PROPERTY PUBLIC LeaderInfo : REFERENCE TO _GVSP_LEADER_PAYLOAD_IMAGE
GET
LeaderInfo REF= _LeaderInfo;
END_GET
END_PROPERTY

PROPERTY PUBLIC LocalIpAddress : REFERENCE TO _UDINT
GET
LocalIpAddress REF= _LocalIpAddress;
END_GET
END_PROPERTY

PROPERTY PUBLIC LocalUdpPort : REFERENCE TO _UINT
GET
LocalUdpPort REF= _LocalUdpPort;
END_GET
END_PROPERTY

METHOD PUBLIC MakeReferenceTo
VAR_INPUT
	ReferenceTarget : REFERENCE TO GVSP_IMAGE_INFO;
END_VAR
activeData REF= ReferenceTarget;
SetMemberReference();
END_METHOD

METHOD PROTECTED SetMemberReference
VAR_INPUT
END_VAR
_CameraIpAddress.MakeReferenceTo(activeData.CameraIpAddress);
_LocalIpAddress.MakeReferenceTo(activeData.LocalIpAddress);
_CameraUdpPort.MakeReferenceTo(activeData.CameraUdpPort);
_LocalUdpPort.MakeReferenceTo(activeData.LocalUdpPort);
_GvspChannelId.MakeReferenceTo(activeData.GvspChannelId);
_GevStatus.MakeReferenceTo(activeData.GevStatus);
_BlockId.MakeReferenceTo(activeData.BlockId);
_LeaderInfo.MakeReferenceTo(activeData.LeaderInfo);
END_METHOD

PROPERTY PUBLIC Size : UDINT
GET
Size := SIZEOF(activeData);
END_GET
END_PROPERTY

METHOD TryMakeReferenceTo : BOOL
VAR_INPUT
	Target : I_Datatype;
END_VAR
VAR
	targetAsStruct : I_StructuredDatatype;
	pTargetData : POINTER TO GVSP_IMAGE_INFO;
END_VAR
IF NOT Target.TryResolveAsStructuredDatatype(targetAsStruct) THEN
	RETURN;
END_IF

IF NOT (targetAsStruct.Identifier = Identifier) THEN
	RETURN;
END_IF

pTargetData := Target.Address;
activeData REF= pTargetData^;
SetMemberReference();
TryMakeReferenceTo := TRUE;
END_METHOD

PROPERTY PUBLIC Value : REFERENCE TO GVSP_IMAGE_INFO
GET
Value REF= activeData;
END_GET
END_PROPERTY

END_FUNCTION_BLOCK

// ---- Datatypes/Structs/_TcVnCodeGradesDM.TcPOU
{attribute 'linkalways'} 
{attribute 'no_explicit_call' := 'This FB is a CLASS and must be accessed using methods or properties'}
{attribute 'enable_dynamic_creation'}
FUNCTION_BLOCK _TcVnCodeGradesDM EXTENDS StructuredDatatypeBase
VAR
	localData : TcVnCodeGradesDM;
	activeData : REFERENCE TO TcVnCodeGradesDM REF= localData;
    _nDecode : _USINT(localdata.nDecode);
    _nSymbolContrast : _USINT(localdata.nSymbolContrast);
    _nModulation : _USINT(localdata.nModulation);
    _nReflectanceMargin : _USINT(localdata.nReflectanceMargin);
    _nFixedPatternDamage : _USINT(localdata.nFixedPatternDamage);
    _nAxialNonuniformity : _USINT(localdata.nAxialNonuniformity);
    _nGridNonuniformity : _USINT(localdata.nGridNonuniformity);
    _nUnusedErrorCorrection : _USINT(localdata.nUnusedErrorCorrection);
    _nOverall : _USINT(localdata.nOverall);
END_VAR

PROPERTY PUBLIC Address : PVOID
GET
Address := ADR(activeData);
END_GET
END_PROPERTY

METHOD PUBLIC ClearReference
VAR_INPUT
END_VAR
activeData REF= localData;
SetMemberReference();
END_METHOD

METHOD PUBLIC Clone : I_Datatype
VAR
    pClone : POINTER TO _TcVnCodeGradesDM;
END_VAR
pClone := __NEW(_TcVnCodeGradesDM());
pClone^.Value := Value;
Clone := pClone^;
END_METHOD

METHOD FB_init : BOOL
VAR_INPUT
	bInitRetains : BOOL; // if TRUE, the retain variables are initialized (warm start / cold start)
	bInCopyCode : BOOL;  // if TRUE, the instance afterwards gets moved into the copy code (online change)
END_VAR
SetMemberReference();
AddMember('nDecode', _nDecode);
AddMember('nSymbolContrast', _nSymbolContrast);
AddMember('nModulation', _nModulation);
AddMember('nReflectanceMargin', _nReflectanceMargin);
AddMember('nFixedPatternDamage', _nFixedPatternDamage);
AddMember('nAxialNonuniformity', _nAxialNonuniformity);
AddMember('nGridNonuniformity', _nGridNonuniformity);
AddMember('nUnusedErrorCorrection', _nUnusedErrorCorrection);
AddMember('nOverall', _nOverall);
END_METHOD

PROPERTY PUBLIC Identifier : T_MAXSTRING
GET
Identifier := 'TcVnCodeGradesDM';
END_GET
END_PROPERTY

METHOD PUBLIC MakeReferenceTo
VAR_INPUT
	ReferenceTarget : REFERENCE TO TcVnCodeGradesDM;
END_VAR
activeData REF= ReferenceTarget;
SetMemberReference();
END_METHOD

PROPERTY PUBLIC nAxialNonuniformity : REFERENCE TO _USINT
GET
nAxialNonuniformity REF= _nAxialNonuniformity;
END_GET
END_PROPERTY

PROPERTY PUBLIC nDecode : REFERENCE TO _USINT
GET
nDecode REF= _nDecode;
END_GET
END_PROPERTY

PROPERTY PUBLIC nFixedPatternDamage : REFERENCE TO _USINT
GET
nFixedPatternDamage REF= _nFixedPatternDamage;
END_GET
END_PROPERTY

PROPERTY PUBLIC nGridNonuniformity : REFERENCE TO _USINT
GET
nGridNonuniformity REF= _nGridNonuniformity;
END_GET
END_PROPERTY

PROPERTY PUBLIC nModulation : REFERENCE TO _USINT
GET
nModulation REF= _nModulation;
END_GET
END_PROPERTY

PROPERTY PUBLIC nOverall : REFERENCE TO _USINT
GET
nOverall REF= _nOverall;
END_GET
END_PROPERTY

PROPERTY PUBLIC nReflectanceMargin : REFERENCE TO _USINT
GET
nReflectanceMargin REF= _nReflectanceMargin;
END_GET
END_PROPERTY

PROPERTY PUBLIC nSymbolContrast : REFERENCE TO _USINT
GET
nSymbolContrast REF= _nSymbolContrast;
END_GET
END_PROPERTY

PROPERTY PUBLIC nUnusedErrorCorrection : REFERENCE TO _USINT
GET
nUnusedErrorCorrection REF= _nUnusedErrorCorrection;
END_GET
END_PROPERTY

METHOD PROTECTED SetMemberReference
VAR_INPUT
END_VAR
_nDecode.MakeReferenceTo(activeData.nDecode);
_nSymbolContrast.MakeReferenceTo(activeData.nSymbolContrast);
_nModulation.MakeReferenceTo(activeData.nModulation);
_nReflectanceMargin.MakeReferenceTo(activeData.nReflectanceMargin);
_nFixedPatternDamage.MakeReferenceTo(activeData.nFixedPatternDamage);
_nAxialNonuniformity.MakeReferenceTo(activeData.nAxialNonuniformity);
_nGridNonuniformity.MakeReferenceTo(activeData.nGridNonuniformity);
_nUnusedErrorCorrection.MakeReferenceTo(activeData.nUnusedErrorCorrection);
_nOverall.MakeReferenceTo(activeData.nOverall);
END_METHOD

PROPERTY PUBLIC Size : UDINT
GET
Size := SIZEOF(activeData);
END_GET
END_PROPERTY

METHOD TryMakeReferenceTo : BOOL
VAR_INPUT
	Target : I_Datatype;
END_VAR
VAR
	pTargetData : POINTER TO TcVnCodeGradesDM;
END_VAR
IF NOT IsEquivalentTo(Target) THEN
	RETURN;
END_IF

pTargetData := Target.Address;
activeData REF= pTargetData^;
SetMemberReference();
TryMakeReferenceTo := TRUE;
END_METHOD

PROPERTY PUBLIC Value : REFERENCE TO TcVnCodeGradesDM
GET
Value REF= activeData;
END_GET
END_PROPERTY

END_FUNCTION_BLOCK

// ---- Datatypes/Structs/_TcVnCodeGradesQR.TcPOU
{attribute 'linkalways'} 
{attribute 'no_explicit_call' := 'This FB is a CLASS and must be accessed using methods or properties'}
{attribute 'enable_dynamic_creation'}
FUNCTION_BLOCK _TcVnCodeGradesQR EXTENDS StructuredDatatypeBase
VAR
	localData : TcVnCodeGradesQR;
	activeData : REFERENCE TO TcVnCodeGradesQR REF= localData;
    _nDecode : _USINT(localdata.nDecode);
    _nSymbolContrast : _USINT(localdata.nSymbolContrast);
    _nModulation : _USINT(localdata.nModulation);
    _nReflectanceMargin : _USINT(localdata.nReflectanceMargin);
    _nFixedPatternDamage : _USINT(localdata.nFixedPatternDamage);
    _nAxialNonuniformity : _USINT(localdata.nAxialNonuniformity);
    _nGridNonuniformity : _USINT(localdata.nGridNonuniformity);
    _nUnusedErrorCorrection : _USINT(localdata.nUnusedErrorCorrection);
    _nFormatInfo : _USINT(localdata.nFormatInfo);
    _nVersionInfo : _USINT(localdata.nVersionInfo);
    _nOverall : _USINT(localdata.nOverall);
END_VAR

PROPERTY PUBLIC Address : PVOID
GET
Address := ADR(activeData);
END_GET
END_PROPERTY

METHOD PUBLIC ClearReference
VAR_INPUT
END_VAR
activeData REF= localData;
SetMemberReference();
END_METHOD

METHOD PUBLIC Clone : I_Datatype
VAR
    pClone : POINTER TO _TcVnCodeGradesQR;
END_VAR
pClone := __NEW(_TcVnCodeGradesQR());
pClone^.Value := Value;
Clone := pClone^;
END_METHOD

METHOD FB_init : BOOL
VAR_INPUT
	bInitRetains : BOOL; // if TRUE, the retain variables are initialized (warm start / cold start)
	bInCopyCode : BOOL;  // if TRUE, the instance afterwards gets moved into the copy code (online change)
END_VAR
SetMemberReference();
AddMember('nDecode', _nDecode);
AddMember('nSymbolContrast', _nSymbolContrast);
AddMember('nModulation', _nModulation);
AddMember('nReflectanceMargin', _nReflectanceMargin);
AddMember('nFixedPatternDamage', _nFixedPatternDamage);
AddMember('nAxialNonuniformity', _nAxialNonuniformity);
AddMember('nGridNonuniformity', _nGridNonuniformity);
AddMember('nUnusedErrorCorrection', _nUnusedErrorCorrection);
AddMember('nFormatInfo', _nFormatInfo);
AddMember('nVersionInfo', _nVersionInfo);
AddMember('nOverall', _nOverall);
END_METHOD

PROPERTY PUBLIC Identifier : T_MAXSTRING
GET
Identifier := 'TcVnCodeGradesQR';
END_GET
END_PROPERTY

METHOD PUBLIC MakeReferenceTo
VAR_INPUT
	ReferenceTarget : REFERENCE TO TcVnCodeGradesQR;
END_VAR
activeData REF= ReferenceTarget;
SetMemberReference();
END_METHOD

PROPERTY PUBLIC nAxialNonuniformity : REFERENCE TO _USINT
GET
nAxialNonuniformity REF= _nAxialNonuniformity;
END_GET
END_PROPERTY

PROPERTY PUBLIC nDecode : REFERENCE TO _USINT
GET
nDecode REF= _nDecode;
END_GET
END_PROPERTY

PROPERTY PUBLIC nFixedPatternDamage : REFERENCE TO _USINT
GET
nFixedPatternDamage REF= _nFixedPatternDamage;
END_GET
END_PROPERTY

PROPERTY PUBLIC nFormatInfo : REFERENCE TO _USINT
GET
nFormatInfo REF= _nFormatInfo;
END_GET
END_PROPERTY

PROPERTY PUBLIC nGridNonuniformity : REFERENCE TO _USINT
GET
nGridNonuniformity REF= _nGridNonuniformity;
END_GET
END_PROPERTY

PROPERTY PUBLIC nModulation : REFERENCE TO _USINT
GET
nModulation REF= _nModulation;
END_GET
END_PROPERTY

PROPERTY PUBLIC nOverall : REFERENCE TO _USINT
GET
nOverall REF= _nOverall;
END_GET
END_PROPERTY

PROPERTY PUBLIC nReflectanceMargin : REFERENCE TO _USINT
GET
nReflectanceMargin REF= _nReflectanceMargin;
END_GET
END_PROPERTY

PROPERTY PUBLIC nSymbolContrast : REFERENCE TO _USINT
GET
nSymbolContrast REF= _nSymbolContrast;
END_GET
END_PROPERTY

PROPERTY PUBLIC nUnusedErrorCorrection : REFERENCE TO _USINT
GET
nUnusedErrorCorrection REF= _nUnusedErrorCorrection;
END_GET
END_PROPERTY

PROPERTY PUBLIC nVersionInfo : REFERENCE TO _USINT
GET
nVersionInfo REF= _nVersionInfo;
END_GET
END_PROPERTY

METHOD PROTECTED SetMemberReference
VAR_INPUT
END_VAR
_nDecode.MakeReferenceTo(activeData.nDecode);
_nSymbolContrast.MakeReferenceTo(activeData.nSymbolContrast);
_nModulation.MakeReferenceTo(activeData.nModulation);
_nReflectanceMargin.MakeReferenceTo(activeData.nReflectanceMargin);
_nFixedPatternDamage.MakeReferenceTo(activeData.nFixedPatternDamage);
_nAxialNonuniformity.MakeReferenceTo(activeData.nAxialNonuniformity);
_nGridNonuniformity.MakeReferenceTo(activeData.nGridNonuniformity);
_nUnusedErrorCorrection.MakeReferenceTo(activeData.nUnusedErrorCorrection);
_nFormatInfo.MakeReferenceTo(activeData.nFormatInfo);
_nVersionInfo.MakeReferenceTo(activeData.nVersionInfo);
_nOverall.MakeReferenceTo(activeData.nOverall);
END_METHOD

PROPERTY PUBLIC Size : UDINT
GET
Size := SIZEOF(activeData);
END_GET
END_PROPERTY

METHOD TryMakeReferenceTo : BOOL
VAR_INPUT
	Target : I_Datatype;
END_VAR
VAR
	pTargetData : POINTER TO TcVnCodeGradesQR;
END_VAR
IF NOT IsEquivalentTo(Target) THEN
	RETURN;
END_IF

pTargetData := Target.Address;
activeData REF= pTargetData^;
SetMemberReference();
TryMakeReferenceTo := TRUE;
END_METHOD

PROPERTY PUBLIC Value : REFERENCE TO TcVnCodeGradesQR
GET
Value REF= activeData;
END_GET
END_PROPERTY

END_FUNCTION_BLOCK

// ---- Datatypes/Structs/_TcVnMoments.TcPOU
{attribute 'linkalways'} 
{attribute 'no_explicit_call' := 'This FB is a CLASS and must be accessed using methods or properties'}
{attribute 'enable_dynamic_creation'}
FUNCTION_BLOCK _TcVnMoments EXTENDS StructuredDatatypeBase
VAR
	localData : TcVnMoments;
	activeData : REFERENCE TO TcVnMoments REF= localData;
    _fM00 : _LREAL(localdata.fM00);
    _fM01 : _LREAL(localdata.fM01);
    _fM02 : _LREAL(localdata.fM02);
    _fM03 : _LREAL(localdata.fM03);
    _fM10 : _LREAL(localdata.fM10);
    _fM11 : _LREAL(localdata.fM11);
    _fM12 : _LREAL(localdata.fM12);
    _fM20 : _LREAL(localdata.fM20);
    _fM21 : _LREAL(localdata.fM21);
    _fM30 : _LREAL(localdata.fM30);
    _fMu02 : _LREAL(localdata.fMu02);
    _fMu03 : _LREAL(localdata.fMu03);
    _fMu11 : _LREAL(localdata.fMu11);
    _fMu12 : _LREAL(localdata.fMu12);
    _fMu20 : _LREAL(localdata.fMu20);
    _fMu21 : _LREAL(localdata.fMu21);
    _fMu30 : _LREAL(localdata.fMu30);
    _fNu02 : _LREAL(localdata.fNu02);
    _fNu03 : _LREAL(localdata.fNu03);
    _fNu11 : _LREAL(localdata.fNu11);
    _fNu12 : _LREAL(localdata.fNu12);
    _fNu20 : _LREAL(localdata.fNu20);
    _fNu21 : _LREAL(localdata.fNu21);
    _fNu30 : _LREAL(localdata.fNu30);
END_VAR

PROPERTY PUBLIC Address : PVOID
GET
Address := ADR(activeData);
END_GET
END_PROPERTY

METHOD PUBLIC ClearReference
VAR_INPUT
END_VAR
activeData REF= localData;
SetMemberReference();
END_METHOD

METHOD PUBLIC Clone : I_Datatype
VAR
    pClone : POINTER TO _TcVnMoments;
END_VAR
pClone := __NEW(_TcVnMoments());
pClone^.Value := Value;
Clone := pClone^;
END_METHOD

METHOD FB_init : BOOL
VAR_INPUT
	bInitRetains : BOOL; // if TRUE, the retain variables are initialized (warm start / cold start)
	bInCopyCode : BOOL;  // if TRUE, the instance afterwards gets moved into the copy code (online change)
END_VAR
SetMemberReference();
AddMember('fM00', _fM00);
AddMember('fM01', _fM01);
AddMember('fM02', _fM02);
AddMember('fM03', _fM03);
AddMember('fM10', _fM10);
AddMember('fM11', _fM11);
AddMember('fM12', _fM12);
AddMember('fM20', _fM20);
AddMember('fM21', _fM21);
AddMember('fM30', _fM30);
AddMember('fMu02', _fMu02);
AddMember('fMu03', _fMu03);
AddMember('fMu11', _fMu11);
AddMember('fMu12', _fMu12);
AddMember('fMu20', _fMu20);
AddMember('fMu21', _fMu21);
AddMember('fMu30', _fMu30);
AddMember('fNu02', _fNu02);
AddMember('fNu03', _fNu03);
AddMember('fNu11', _fNu11);
AddMember('fNu12', _fNu12);
AddMember('fNu20', _fNu20);
AddMember('fNu21', _fNu21);
AddMember('fNu30', _fNu30);
END_METHOD

PROPERTY PUBLIC fM00 : REFERENCE TO _LREAL
GET
fM00 REF= _fM00;
END_GET
END_PROPERTY

PROPERTY PUBLIC fM01 : REFERENCE TO _LREAL
GET
fM01 REF= _fM01;
END_GET
END_PROPERTY

PROPERTY PUBLIC fM02 : REFERENCE TO _LREAL
GET
fM02 REF= _fM02;
END_GET
END_PROPERTY

PROPERTY PUBLIC fM03 : REFERENCE TO _LREAL
GET
fM03 REF= _fM03;
END_GET
END_PROPERTY

PROPERTY PUBLIC fM10 : REFERENCE TO _LREAL
GET
fM10 REF= _fM10;
END_GET
END_PROPERTY

PROPERTY PUBLIC fM11 : REFERENCE TO _LREAL
GET
fM11 REF= _fM11;
END_GET
END_PROPERTY

PROPERTY PUBLIC fM12 : REFERENCE TO _LREAL
GET
fM12 REF= _fM12;
END_GET
END_PROPERTY

PROPERTY PUBLIC fM20 : REFERENCE TO _LREAL
GET
fM20 REF= _fM20;
END_GET
END_PROPERTY

PROPERTY PUBLIC fM21 : REFERENCE TO _LREAL
GET
fM21 REF= _fM21;
END_GET
END_PROPERTY

PROPERTY PUBLIC fM30 : REFERENCE TO _LREAL
GET
fM30 REF= _fM30;
END_GET
END_PROPERTY

PROPERTY PUBLIC fMu02 : REFERENCE TO _LREAL
GET
fMu02 REF= _fMu02;
END_GET
END_PROPERTY

PROPERTY PUBLIC fMu03 : REFERENCE TO _LREAL
GET
fMu03 REF= _fMu03;
END_GET
END_PROPERTY

PROPERTY PUBLIC fMu11 : REFERENCE TO _LREAL
GET
fMu11 REF= _fMu11;
END_GET
END_PROPERTY

PROPERTY PUBLIC fMu12 : REFERENCE TO _LREAL
GET
fMu12 REF= _fMu12;
END_GET
END_PROPERTY

PROPERTY PUBLIC fMu20 : REFERENCE TO _LREAL
GET
fMu20 REF= _fMu20;
END_GET
END_PROPERTY

PROPERTY PUBLIC fMu21 : REFERENCE TO _LREAL
GET
fMu21 REF= _fMu21;
END_GET
END_PROPERTY

PROPERTY PUBLIC fMu30 : REFERENCE TO _LREAL
GET
fMu30 REF= _fMu30;
END_GET
END_PROPERTY

PROPERTY PUBLIC fNu02 : REFERENCE TO _LREAL
GET
fNu02 REF= _fNu02;
END_GET
END_PROPERTY

PROPERTY PUBLIC fNu03 : REFERENCE TO _LREAL
GET
fNu03 REF= _fNu03;
END_GET
END_PROPERTY

PROPERTY PUBLIC fNu11 : REFERENCE TO _LREAL
GET
fNu11 REF= _fNu11;
END_GET
END_PROPERTY

PROPERTY PUBLIC fNu12 : REFERENCE TO _LREAL
GET
fNu12 REF= _fNu12;
END_GET
END_PROPERTY

PROPERTY PUBLIC fNu20 : REFERENCE TO _LREAL
GET
fNu20 REF= _fNu20;
END_GET
END_PROPERTY

PROPERTY PUBLIC fNu21 : REFERENCE TO _LREAL
GET
fNu21 REF= _fNu21;
END_GET
END_PROPERTY

PROPERTY PUBLIC fNu30 : REFERENCE TO _LREAL
GET
fNu30 REF= _fNu30;
END_GET
END_PROPERTY

PROPERTY PUBLIC Identifier : T_MAXSTRING
GET
Identifier := 'TcVnMoments';
END_GET
END_PROPERTY

METHOD PUBLIC MakeReferenceTo
VAR_INPUT
	ReferenceTarget : REFERENCE TO TcVnMoments;
END_VAR
activeData REF= ReferenceTarget;
SetMemberReference();
END_METHOD

METHOD PROTECTED SetMemberReference
VAR_INPUT
END_VAR
_fM00.MakeReferenceTo(activeData.fM00);
_fM01.MakeReferenceTo(activeData.fM01);
_fM02.MakeReferenceTo(activeData.fM02);
_fM03.MakeReferenceTo(activeData.fM03);
_fM10.MakeReferenceTo(activeData.fM10);
_fM11.MakeReferenceTo(activeData.fM11);
_fM12.MakeReferenceTo(activeData.fM12);
_fM20.MakeReferenceTo(activeData.fM20);
_fM21.MakeReferenceTo(activeData.fM21);
_fM30.MakeReferenceTo(activeData.fM30);
_fMu02.MakeReferenceTo(activeData.fMu02);
_fMu03.MakeReferenceTo(activeData.fMu03);
_fMu11.MakeReferenceTo(activeData.fMu11);
_fMu12.MakeReferenceTo(activeData.fMu12);
_fMu20.MakeReferenceTo(activeData.fMu20);
_fMu21.MakeReferenceTo(activeData.fMu21);
_fMu30.MakeReferenceTo(activeData.fMu30);
_fNu02.MakeReferenceTo(activeData.fNu02);
_fNu03.MakeReferenceTo(activeData.fNu03);
_fNu11.MakeReferenceTo(activeData.fNu11);
_fNu12.MakeReferenceTo(activeData.fNu12);
_fNu20.MakeReferenceTo(activeData.fNu20);
_fNu21.MakeReferenceTo(activeData.fNu21);
_fNu30.MakeReferenceTo(activeData.fNu30);
END_METHOD

PROPERTY PUBLIC Size : UDINT
GET
Size := SIZEOF(activeData);
END_GET
END_PROPERTY

METHOD TryMakeReferenceTo : BOOL
VAR_INPUT
	Target : I_Datatype;
END_VAR
VAR
	pTargetData : POINTER TO TcVnMoments;
END_VAR
IF NOT IsEquivalentTo(Target) THEN
	RETURN;
END_IF

pTargetData := Target.Address;
activeData REF= pTargetData^;
SetMemberReference();
TryMakeReferenceTo := TRUE;
END_METHOD

PROPERTY PUBLIC Value : REFERENCE TO TcVnMoments
GET
Value REF= activeData;
END_GET
END_PROPERTY

END_FUNCTION_BLOCK

// ---- Datatypes/Structs/_TcVnDMatch.TcPOU
{attribute 'linkalways'} 
{attribute 'no_explicit_call' := 'This FB is a CLASS and must be accessed using methods or properties'}
{attribute 'enable_dynamic_creation'}
FUNCTION_BLOCK _TcVnDMatch EXTENDS StructuredDatatypeBase
VAR
	localData : TcVnDMatch;
	activeData : REFERENCE TO TcVnDMatch REF= localData;
    _nQueryIdx : _DINT(localdata.nQueryIdx);
    _nTrainIdx : _DINT(localdata.nTrainIdx);
    _nImageIdx : _DINT(localdata.nImageIdx);
    _fDistance : _REAL(localdata.fDistance);
END_VAR

PROPERTY PUBLIC Address : PVOID
GET
Address := ADR(activeData);
END_GET
END_PROPERTY

METHOD PUBLIC ClearReference
VAR_INPUT
END_VAR
activeData REF= localData;
SetMemberReference();
END_METHOD

METHOD PUBLIC Clone : I_Datatype
VAR
    pClone : POINTER TO _TcVnDMatch;
END_VAR
pClone := __NEW(_TcVnDMatch());
pClone^.Value := Value;
Clone := pClone^;
END_METHOD

METHOD FB_init : BOOL
VAR_INPUT
	bInitRetains : BOOL; // if TRUE, the retain variables are initialized (warm start / cold start)
	bInCopyCode : BOOL;  // if TRUE, the instance afterwards gets moved into the copy code (online change)
END_VAR
SetMemberReference();
AddMember('nQueryIdx', _nQueryIdx);
AddMember('nTrainIdx', _nTrainIdx);
AddMember('nImageIdx', _nImageIdx);
AddMember('fDistance', _fDistance);
END_METHOD

PROPERTY PUBLIC fDistance : REFERENCE TO _REAL
GET
fDistance REF= _fDistance;
END_GET
END_PROPERTY

PROPERTY PUBLIC Identifier : T_MAXSTRING
GET
Identifier := 'TcVnDMatch';
END_GET
END_PROPERTY

METHOD PUBLIC MakeReferenceTo
VAR_INPUT
	ReferenceTarget : REFERENCE TO TcVnDMatch;
END_VAR
activeData REF= ReferenceTarget;
SetMemberReference();
END_METHOD

PROPERTY PUBLIC nImageIdx : REFERENCE TO _DINT
GET
nImageIdx REF= _nImageIdx;
END_GET
END_PROPERTY

PROPERTY PUBLIC nQueryIdx : REFERENCE TO _DINT
GET
nQueryIdx REF= _nQueryIdx;
END_GET
END_PROPERTY

PROPERTY PUBLIC nTrainIdx : REFERENCE TO _DINT
GET
nTrainIdx REF= _nTrainIdx;
END_GET
END_PROPERTY

METHOD PROTECTED SetMemberReference
VAR_INPUT
END_VAR
_nQueryIdx.MakeReferenceTo(activeData.nQueryIdx);
_nTrainIdx.MakeReferenceTo(activeData.nTrainIdx);
_nImageIdx.MakeReferenceTo(activeData.nImageIdx);
_fDistance.MakeReferenceTo(activeData.fDistance);
END_METHOD

PROPERTY PUBLIC Size : UDINT
GET
Size := SIZEOF(activeData);
END_GET
END_PROPERTY

METHOD TryMakeReferenceTo : BOOL
VAR_INPUT
	Target : I_Datatype;
END_VAR
VAR
	targetAsStruct : I_StructuredDatatype;
	pTargetData : POINTER TO TcVnDMatch;
END_VAR
IF NOT Target.TryResolveAsStructuredDatatype(targetAsStruct) THEN
	RETURN;
END_IF

IF NOT (targetAsStruct.Identifier = Identifier) THEN
	RETURN;
END_IF

pTargetData := Target.Address;
activeData REF= pTargetData^;
SetMemberReference();
TryMakeReferenceTo := TRUE;
END_METHOD

PROPERTY PUBLIC Value : REFERENCE TO TcVnDMatch
GET
Value REF= activeData;
END_GET
END_PROPERTY

END_FUNCTION_BLOCK

// ---- Datatypes/Structs/_TcVnCodeGrades1D.TcPOU
{attribute 'linkalways'} 
{attribute 'no_explicit_call' := 'This FB is a CLASS and must be accessed using methods or properties'}
{attribute 'enable_dynamic_creation'}
FUNCTION_BLOCK _TcVnCodeGrades1D EXTENDS StructuredDatatypeBase
VAR
	localData : TcVnCodeGrades1D;
	activeData : REFERENCE TO TcVnCodeGrades1D REF= localData;
    _fDecode : _REAL(localdata.fDecode);
    _fSymbolContrast : _REAL(localdata.fSymbolContrast);
    _fMinReflectance : _REAL(localdata.fMinReflectance);
    _fMinEdgeContrast : _REAL(localdata.fMinEdgeContrast);
    _fModulation : _REAL(localdata.fModulation);
    _fDefects : _REAL(localdata.fDefects);
    _fDecodability : _REAL(localdata.fDecodability);
    _fOverall : _REAL(localdata.fOverall);
END_VAR

PROPERTY PUBLIC Address : PVOID
GET
Address := ADR(activeData);
END_GET
END_PROPERTY

METHOD PUBLIC ClearReference
VAR_INPUT
END_VAR
activeData REF= localData;
SetMemberReference();
END_METHOD

METHOD PUBLIC Clone : I_Datatype
VAR
    pClone : POINTER TO _TcVnCodeGrades1D;
END_VAR
pClone := __NEW(_TcVnCodeGrades1D());
pClone^.Value := Value;
Clone := pClone^;
END_METHOD

METHOD FB_init : BOOL
VAR_INPUT
	bInitRetains : BOOL; // if TRUE, the retain variables are initialized (warm start / cold start)
	bInCopyCode : BOOL;  // if TRUE, the instance afterwards gets moved into the copy code (online change)
END_VAR
SetMemberReference();
AddMember('fDecode', _fDecode);
AddMember('fSymbolContrast', _fSymbolContrast);
AddMember('fMinReflectance', _fMinReflectance);
AddMember('fMinEdgeContrast', _fMinEdgeContrast);
AddMember('fModulation', _fModulation);
AddMember('fDefects', _fDefects);
AddMember('fDecodability', _fDecodability);
AddMember('fOverall', _fOverall);
END_METHOD

PROPERTY PUBLIC fDecodability : REFERENCE TO _REAL
GET
fDecodability REF= _fDecodability;
END_GET
END_PROPERTY

PROPERTY PUBLIC fDecode : REFERENCE TO _REAL
GET
fDecode REF= _fDecode;
END_GET
END_PROPERTY

PROPERTY PUBLIC fDefects : REFERENCE TO _REAL
GET
fDefects REF= _fDefects;
END_GET
END_PROPERTY

PROPERTY PUBLIC fMinEdgeContrast : REFERENCE TO _REAL
GET
fMinEdgeContrast REF= _fMinEdgeContrast;
END_GET
END_PROPERTY

PROPERTY PUBLIC fMinReflectance : REFERENCE TO _REAL
GET
fMinReflectance REF= _fMinReflectance;
END_GET
END_PROPERTY

PROPERTY PUBLIC fModulation : REFERENCE TO _REAL
GET
fModulation REF= _fModulation;
END_GET
END_PROPERTY

PROPERTY PUBLIC fOverall : REFERENCE TO _REAL
GET
fOverall REF= _fOverall;
END_GET
END_PROPERTY

PROPERTY PUBLIC fSymbolContrast : REFERENCE TO _REAL
GET
fSymbolContrast REF= _fSymbolContrast;
END_GET
END_PROPERTY

PROPERTY PUBLIC Identifier : T_MAXSTRING
GET
Identifier := 'TcVnCodeGrades1D';
END_GET
END_PROPERTY

METHOD PUBLIC MakeReferenceTo
VAR_INPUT
	ReferenceTarget : REFERENCE TO TcVnCodeGrades1D;
END_VAR
activeData REF= ReferenceTarget;
SetMemberReference();
END_METHOD

METHOD PROTECTED SetMemberReference
VAR_INPUT
END_VAR
_fDecode.MakeReferenceTo(activeData.fDecode);
_fSymbolContrast.MakeReferenceTo(activeData.fSymbolContrast);
_fMinReflectance.MakeReferenceTo(activeData.fMinReflectance);
_fMinEdgeContrast.MakeReferenceTo(activeData.fMinEdgeContrast);
_fModulation.MakeReferenceTo(activeData.fModulation);
_fDefects.MakeReferenceTo(activeData.fDefects);
_fDecodability.MakeReferenceTo(activeData.fDecodability);
_fOverall.MakeReferenceTo(activeData.fOverall);
END_METHOD

PROPERTY PUBLIC Size : UDINT
GET
Size := SIZEOF(activeData);
END_GET
END_PROPERTY

METHOD TryMakeReferenceTo : BOOL
VAR_INPUT
	Target : I_Datatype;
END_VAR
VAR
	pTargetData : POINTER TO TcVnCodeGrades1D;
END_VAR
IF NOT IsEquivalentTo(Target) THEN
	RETURN;
END_IF

pTargetData := Target.Address;
activeData REF= pTargetData^;
SetMemberReference();
TryMakeReferenceTo := TRUE;
END_METHOD

PROPERTY PUBLIC Value : REFERENCE TO TcVnCodeGrades1D
GET
Value REF= activeData;
END_GET
END_PROPERTY

END_FUNCTION_BLOCK

// ---- Datatypes/Structs/_TcVnMatrix.TcPOU
{attribute 'linkalways'} 
{attribute 'no_explicit_call' := 'This FB is a CLASS and must be accessed using methods or properties'}
{attribute 'enable_dynamic_creation'}
FUNCTION_BLOCK _TcVnMatrix EXTENDS StructuredDatatypeBase
VAR
	localData : TcVnMatrix;
	activeData : REFERENCE TO TcVnMatrix REF= localData;
	_nRows : _UDINT(localData.nRows);
    _nCols : _UDINT(localData.nCols);
    _eType : _ETcVnElementType(localData.eType);
    _pData : _PVOID(localData.pData);
END_VAR

PROPERTY PUBLIC Address : PVOID
GET
Address := ADR(activeData);
END_GET
END_PROPERTY

METHOD PUBLIC ClearReference
VAR_INPUT
END_VAR
activeData REF= localData;
SetMemberReference();
END_METHOD

METHOD PUBLIC Clone : I_Datatype
VAR
    pClone : POINTER TO _TcVnMatrix;
END_VAR
pClone := __NEW(_TcVnMatrix());
pClone^.Value := Value;
Clone := pClone^;
END_METHOD

PROPERTY PUBLIC eType : REFERENCE TO _ETcVnElementType
GET
eType REF= _eType;
END_GET
END_PROPERTY

METHOD FB_init : BOOL
VAR_INPUT
	bInitRetains : BOOL; // if TRUE, the retain variables are initialized (warm start / cold start)
	bInCopyCode : BOOL;  // if TRUE, the instance afterwards gets moved into the copy code (online change)
END_VAR
SetMemberReference();
AddMember('nRows', _nRows);
AddMember('nCols', _nCols);
AddMember('eType', _eType);
AddMember('pData', _pData);
END_METHOD

PROPERTY PUBLIC Identifier : T_MAXSTRING
GET
Identifier := 'TcVnMatrix';
END_GET
END_PROPERTY

METHOD PUBLIC MakeReferenceTo
VAR_INPUT
	ReferenceTarget : REFERENCE TO TcVnMatrix;
END_VAR
activeData REF= ReferenceTarget;
SetMemberReference();
END_METHOD

PROPERTY PUBLIC nCols : REFERENCE TO _UDINT
GET
nCols REF= _nCols;
END_GET
END_PROPERTY

PROPERTY PUBLIC nRows : REFERENCE TO _UDINT
GET
nRows REF= _nRows;
END_GET
END_PROPERTY

PROPERTY PUBLIC pData : REFERENCE TO _PVOID
GET
pData REF= _pData;
END_GET
END_PROPERTY

METHOD PROTECTED SetMemberReference
VAR_INPUT
END_VAR
_nRows.MakeReferenceTo(activeData.nRows);
_nCols.MakeReferenceTo(activeData.nCols);
_eType.MakeReferenceTo(activeData.eType);
_pData.MakeReferenceTo(activeData.pData);
END_METHOD

PROPERTY PUBLIC Size : UDINT
GET
Size := SIZEOF(activeData);
END_GET
END_PROPERTY

METHOD TryMakeReferenceTo : BOOL
VAR_INPUT
	Target : I_Datatype;
END_VAR
VAR
	pTargetData : POINTER TO TcVnMatrix;
END_VAR
IF NOT IsEquivalentTo(Target) THEN
	RETURN;
END_IF

pTargetData := Target.Address;
activeData REF= pTargetData^;
SetMemberReference();
TryMakeReferenceTo := TRUE;
END_METHOD

PROPERTY PUBLIC Value : REFERENCE TO TcVnMatrix
GET
Value REF= activeData;
END_GET
END_PROPERTY

END_FUNCTION_BLOCK

// ---- Datatypes/Structs/_TcVnParamsMSER.TcPOU
{attribute 'linkalways'} 
{attribute 'no_explicit_call' := 'This FB is a CLASS and must be accessed using methods or properties'}
{attribute 'enable_dynamic_creation'}
FUNCTION_BLOCK _TcVnParamsMSER EXTENDS StructuredDatatypeBase
VAR
	localData : TcVnParamsMSER;
	activeData : REFERENCE TO TcVnParamsMSER REF= localData;
	_nDelta : _DINT(localData.nDelta);
    _nMinArea : _UDINT(localData.nMinArea);
	_nMaxArea : _UDINT(localData.nMaxArea);
	_fMaxVariation : _LREAL(localData.fMaxVariation);
	_fMinDiversity : _LREAL(localData.fMinDiversity);
	_nMaxEvolution : _UDINT(localData.nMaxEvolution);
    _fAreaThreshold : _LREAL(localData.fAreaThreshold);
    _fMinMargin : _LREAL(localData.fMinMargin);
    _nEdgeBlurSize : _UDINT(localData.nEdgeBlurSize);
END_VAR

PROPERTY PUBLIC Address : PVOID
GET
Address := ADR(activeData);
END_GET
END_PROPERTY

METHOD PUBLIC ClearReference
VAR_INPUT
END_VAR
activeData REF= localData;
SetMemberReference();
END_METHOD

METHOD PUBLIC Clone : I_Datatype
VAR
    pClone : POINTER TO _TcVnParamsMSER;
END_VAR
pClone := __NEW(_TcVnParamsMSER());
pClone^.Value := Value;
Clone := pClone^;
END_METHOD

PROPERTY PUBLIC fAreaThreshold : REFERENCE TO _LREAL
GET
fAreaThreshold REF= _fAreaThreshold;
END_GET
END_PROPERTY

METHOD FB_init : BOOL
VAR_INPUT
	bInitRetains : BOOL; // if TRUE, the retain variables are initialized (warm start / cold start)
	bInCopyCode : BOOL;  // if TRUE, the instance afterwards gets moved into the copy code (online change)
END_VAR
SetMemberReference();
AddMember('nDelta', _nDelta);
AddMember('nMinArea', _nMinArea);
AddMember('nMaxArea', _nMaxArea);
AddMember('fMaxVariation', _fMaxVariation);
AddMember('fMinDiversity', _fMinDiversity);
AddMember('nMaxEvolution', _nMaxEvolution);
AddMember('fAreaThreshold', _fAreaThreshold);
AddMember('fMinMargin', _fMinMargin);
AddMember('nEdgeBlurSize', _nEdgeBlurSize);
END_METHOD

PROPERTY PUBLIC fMaxVariation : REFERENCE TO _LREAL
GET
fMaxVariation REF= _fMaxVariation;
END_GET
END_PROPERTY

PROPERTY PUBLIC fMinDiversity : REFERENCE TO _LREAL
GET
fMinDiversity REF= _fMinDiversity;
END_GET
END_PROPERTY

PROPERTY PUBLIC fMinMargin : REFERENCE TO _LREAL
GET
fMinMargin REF= _fMinMargin;
END_GET
END_PROPERTY

PROPERTY PUBLIC Identifier : T_MAXSTRING
GET
Identifier := 'TcVnParamsMSER';
END_GET
END_PROPERTY

METHOD PUBLIC MakeReferenceTo
VAR_INPUT
	ReferenceTarget : REFERENCE TO TcVnParamsMSER;
END_VAR
activeData REF= ReferenceTarget;
SetMemberReference();
END_METHOD

PROPERTY PUBLIC nDelta : REFERENCE TO _DINT
GET
nDelta REF= _nDelta;
END_GET
END_PROPERTY

PROPERTY PUBLIC nEdgeBlurSize : REFERENCE TO _UDINT
GET
nEdgeBlurSize REF= _nEdgeBlurSize;
END_GET
END_PROPERTY

PROPERTY PUBLIC nMaxArea : REFERENCE TO _UDINT
GET
nMaxArea REF= _nMaxArea;
END_GET
END_PROPERTY

PROPERTY PUBLIC nMaxEvolution : REFERENCE TO _UDINT
GET
nMaxEvolution REF= _nMaxEvolution;
END_GET
END_PROPERTY

PROPERTY PUBLIC nMinArea : REFERENCE TO _UDINT
GET
nMinArea REF= _nMinArea;
END_GET
END_PROPERTY

METHOD PROTECTED SetMemberReference
VAR_INPUT
END_VAR
_nDelta.MakeReferenceTo(activeData.nDelta);
_nMinArea.MakeReferenceTo(activeData.nMinArea);
_nMaxArea.MakeReferenceTo(activeData.nMaxArea);
_fMaxVariation.MakeReferenceTo(activeData.fMaxVariation);
_fMinDiversity.MakeReferenceTo(activeData.fMinDiversity);
_nMaxEvolution.MakeReferenceTo(activeData.nMaxEvolution);
_fAreaThreshold.MakeReferenceTo(activeData.fAreaThreshold);
_fMinMargin.MakeReferenceTo(activeData.fMinMargin);
_nEdgeBlurSize.MakeReferenceTo(activeData.nEdgeBlurSize);
END_METHOD

PROPERTY PUBLIC Size : UDINT
GET
Size := SIZEOF(activeData);
END_GET
END_PROPERTY

METHOD TryMakeReferenceTo : BOOL
VAR_INPUT
	Target : I_Datatype;
END_VAR
VAR
	pTargetData : POINTER TO TcVnParamsMSER;
END_VAR
IF NOT IsEquivalentTo(Target) THEN
	RETURN;
END_IF

pTargetData := Target.Address;
activeData REF= pTargetData^;
SetMemberReference();
TryMakeReferenceTo := TRUE;
END_METHOD

PROPERTY PUBLIC Value : REFERENCE TO TcVnParamsMSER
GET
Value REF= activeData;
END_GET
END_PROPERTY

END_FUNCTION_BLOCK

// ---- Datatypes/Structs/_TcVnParamsAKAZE.TcPOU
{attribute 'linkalways'} 
{attribute 'no_explicit_call' := 'This FB is a CLASS and must be accessed using methods or properties'}
{attribute 'enable_dynamic_creation'}
FUNCTION_BLOCK _TcVnParamsAKAZE EXTENDS StructuredDatatypeBase
VAR
	localData : TcVnParamsAKAZE;
	activeData : REFERENCE TO TcVnParamsAKAZE REF= localData;
    _eDescrType     : _ETcVnFeatureDescriptorTypeAKAZE(localdata.eDescrType);
    _nDescrSize     : _UDINT(localdata.nDescrSize);
    _nDescrChannels : _UDINT(localdata.nDescrChannels);
    _fThreshold     : _REAL(localdata.fThreshold);
    _nOctaves       : _UDINT(localdata.nOctaves);
    _nOctaveLayers  : _UDINT(localdata.nOctaveLayers);
    _eDiffusivity   : _ETcVnDiffusivityTypeKAZE(localdata.eDiffusivity);
END_VAR

PROPERTY PUBLIC Address : PVOID
GET
Address := ADR(activeData);
END_GET
END_PROPERTY

METHOD PUBLIC ClearReference
VAR_INPUT
END_VAR
activeData REF= localData;
SetMemberReference();
END_METHOD

METHOD PUBLIC Clone : I_Datatype
VAR
    pClone : POINTER TO _TcVnParamsAKAZE;
END_VAR
pClone := __NEW(_TcVnParamsAKAZE());
pClone^.Value := Value;
Clone := pClone^;
END_METHOD

PROPERTY PUBLIC eDescrType : REFERENCE TO _ETcVnFeatureDescriptorTypeAKAZE
GET
eDescrType REF= _eDescrType;
END_GET
END_PROPERTY

PROPERTY PUBLIC eDiffusivity : REFERENCE TO _ETcVnDiffusivityTypeKAZE
GET
eDiffusivity REF= _eDiffusivity;
END_GET
END_PROPERTY

METHOD FB_init : BOOL
VAR_INPUT
	bInitRetains : BOOL; // if TRUE, the retain variables are initialized (warm start / cold start)
	bInCopyCode : BOOL;  // if TRUE, the instance afterwards gets moved into the copy code (online change)
END_VAR
SetMemberReference();
AddMember('eDescrType', _eDescrType);
AddMember('nDescrSize', _nDescrSize);
AddMember('nDescrChannels', _nDescrChannels);
AddMember('fThreshold', _fThreshold);
AddMember('nOctaves', _nOctaves);
AddMember('nOctaveLayers', _nOctaveLayers);
AddMember('eDiffusivity', _eDiffusivity);
END_METHOD

PROPERTY PUBLIC fThreshold : REFERENCE TO _REAL
GET
fThreshold REF= _fThreshold;
END_GET
END_PROPERTY

PROPERTY PUBLIC Identifier : T_MAXSTRING
GET
Identifier := 'TcVnParamsAKAZE';
END_GET
END_PROPERTY

METHOD PUBLIC MakeReferenceTo
VAR_INPUT
	ReferenceTarget : REFERENCE TO TcVnParamsAKAZE;
END_VAR
activeData REF= ReferenceTarget;
SetMemberReference();
END_METHOD

PROPERTY PUBLIC nDescrChannels : REFERENCE TO _UDINT
GET
nDescrChannels REF= _nDescrChannels;
END_GET
END_PROPERTY

PROPERTY PUBLIC nDescrSize : REFERENCE TO _UDINT
GET
nDescrSize REF= _nDescrSize;
END_GET
END_PROPERTY

PROPERTY PUBLIC nOctaveLayers : REFERENCE TO _UDINT
GET
nOctaveLayers REF= _nOctaveLayers;
END_GET
END_PROPERTY

PROPERTY PUBLIC nOctaves : REFERENCE TO _UDINT
GET
nOctaves REF= _nOctaves;
END_GET
END_PROPERTY

METHOD PROTECTED SetMemberReference
VAR_INPUT
END_VAR
_eDescrType.MakeReferenceTo(activeData.eDescrType);
_nDescrSize.MakeReferenceTo(activeData.nDescrSize);
_nDescrChannels.MakeReferenceTo(activeData.nDescrChannels);
_fThreshold.MakeReferenceTo(activeData.fThreshold);
_nOctaves.MakeReferenceTo(activeData.nOctaves);
_nOctaveLayers.MakeReferenceTo(activeData.nOctaveLayers);
_eDiffusivity.MakeReferenceTo(activeData.eDiffusivity);
END_METHOD

PROPERTY PUBLIC Size : UDINT
GET
Size := SIZEOF(activeData);
END_GET
END_PROPERTY

METHOD TryMakeReferenceTo : BOOL
VAR_INPUT
	Target : I_Datatype;
END_VAR
VAR
	pTargetData : POINTER TO TcVnParamsAKAZE;
END_VAR
IF NOT IsEquivalentTo(Target) THEN
	RETURN;
END_IF

pTargetData := Target.Address;
activeData REF= pTargetData^;
SetMemberReference();
TryMakeReferenceTo := TRUE;
END_METHOD

PROPERTY PUBLIC Value : REFERENCE TO TcVnParamsAKAZE
GET
Value REF= activeData;
END_GET
END_PROPERTY

END_FUNCTION_BLOCK

// ---- Datatypes/Structs/_TcVnParamsSB.TcPOU
{attribute 'linkalways'} 
{attribute 'no_explicit_call' := 'This FB is a CLASS and must be accessed using methods or properties'}
{attribute 'enable_dynamic_creation'}
FUNCTION_BLOCK _TcVnParamsSB EXTENDS StructuredDatatypeBase
VAR
	localData : TcVnParamsSB;
	activeData : REFERENCE TO TcVnParamsSB REF= localData;
    _bFilterByArea         : _BOOL(localdata.bFilterByArea);
    _bFilterByCircularity  : _BOOL(localdata.bFilterByCircularity);
    _bFilterByColor        : _BOOL(localdata.bFilterByColor);
    _bFilterByConvexity    : _BOOL(localdata.bFilterByConvexity);
    _bFilterByInertia      : _BOOL(localdata.bFilterByInertia);
    _fMinArea              : _REAL(localdata.fMinArea);
    _fMaxArea              : _REAL(localdata.fMaxArea);
    _fMinCircularity       : _REAL(localdata.fMinCircularity);
    _fMaxCircularity       : _REAL(localdata.fMaxCircularity);
    _nBlobColor            : _USINT(localdata.nBlobColor);
    _fMinConvexity         : _REAL(localdata.fMinConvexity);
    _fMaxConvexity         : _REAL(localdata.fMaxConvexity);
    _fMinInertiaRatio      : _REAL(localdata.fMinInertiaRatio);
    _fMaxInertiaRatio      : _REAL(localdata.fMaxInertiaRatio);
    _fMinBlobDist          : _REAL(localdata.fMinBlobDist);
    _nMinRepeatability     : _UDINT(localdata.nMinRepeatability);
    _fMinThreshold         : _REAL(localdata.fMinThreshold);
    _fMaxThreshold         : _REAL(localdata.fMaxThreshold);
    _fThresholdStep        : _REAL(localdata.fThresholdStep);
END_VAR

PROPERTY PUBLIC Address : PVOID
GET
Address := ADR(activeData);
END_GET
END_PROPERTY

PROPERTY PUBLIC bFilterByArea : REFERENCE TO _BOOL
GET
bFilterByArea REF= _bFilterByArea;
END_GET
END_PROPERTY

PROPERTY PUBLIC bFilterByCircularity : REFERENCE TO _BOOL
GET
bFilterByCircularity REF= _bFilterByCircularity;
END_GET
END_PROPERTY

PROPERTY PUBLIC bFilterByColor : REFERENCE TO _BOOL
GET
bFilterByColor REF= _bFilterByColor;
END_GET
END_PROPERTY

PROPERTY PUBLIC bFilterByConvexity : REFERENCE TO _BOOL
GET
bFilterByConvexity REF= _bFilterByConvexity;
END_GET
END_PROPERTY

PROPERTY PUBLIC bFilterByInertia : REFERENCE TO _BOOL
GET
bFilterByInertia REF= _bFilterByInertia;
END_GET
END_PROPERTY

METHOD PUBLIC ClearReference
VAR_INPUT
END_VAR
activeData REF= localData;
SetMemberReference();
END_METHOD

METHOD PUBLIC Clone : I_Datatype
VAR
    pClone : POINTER TO _TcVnParamsSB;
END_VAR
pClone := __NEW(_TcVnParamsSB());
pClone^.Value := Value;
Clone := pClone^;
END_METHOD

METHOD FB_init : BOOL
VAR_INPUT
	bInitRetains : BOOL; // if TRUE, the retain variables are initialized (warm start / cold start)
	bInCopyCode : BOOL;  // if TRUE, the instance afterwards gets moved into the copy code (online change)
END_VAR
SetMemberReference();
AddMember('bFilterByArea', _bFilterByArea);
AddMember('bFilterByCircularity', _bFilterByCircularity);
AddMember('bFilterByColor', _bFilterByColor);
AddMember('bFilterByConvexity', _bFilterByConvexity);
AddMember('bFilterByInertia', _bFilterByInertia);
AddMember('fMinArea', _fMinArea);
AddMember('fMaxArea', _fMaxArea);
AddMember('fMinCircularity', _fMinCircularity);
AddMember('fMaxCircularity', _fMaxCircularity);
AddMember('nBlobColor', _nBlobColor);
AddMember('fMinConvexity', _fMinConvexity);
AddMember('fMaxConvexity', _fMaxConvexity);
AddMember('fMinInertiaRatio', _fMinInertiaRatio);
AddMember('fMaxInertiaRatio', _fMaxInertiaRatio);
AddMember('fMinBlobDist', _fMinBlobDist);
AddMember('nMinRepeatability', _nMinRepeatability);
AddMember('fMinThreshold', _fMinThreshold);
AddMember('fMaxThreshold', _fMaxThreshold);
AddMember('fThresholdStep',  _fThresholdStep);
END_METHOD

PROPERTY PUBLIC fMaxArea : REFERENCE TO _REAL
GET
fMaxArea REF= _fMaxArea;
END_GET
END_PROPERTY

PROPERTY PUBLIC fMaxCircularity : REFERENCE TO _REAL
GET
fMaxCircularity REF= _fMaxCircularity;
END_GET
END_PROPERTY

PROPERTY PUBLIC fMaxConvexity : REFERENCE TO _REAL
GET
fMaxConvexity REF= _fMaxConvexity;
END_GET
END_PROPERTY

PROPERTY PUBLIC fMaxInertiaRatio : REFERENCE TO _REAL
GET
fMaxInertiaRatio REF= _fMaxInertiaRatio;
END_GET
END_PROPERTY

PROPERTY PUBLIC fMaxThreshold : REFERENCE TO _REAL
GET
fMaxThreshold REF= _fMaxThreshold;
END_GET
END_PROPERTY

PROPERTY PUBLIC fMinArea : REFERENCE TO _REAL
GET
fMinArea REF= _fMinArea;
END_GET
END_PROPERTY

PROPERTY PUBLIC fMinBlobDist : REFERENCE TO _REAL
GET
fMinBlobDist REF= _fMinBlobDist;
END_GET
END_PROPERTY

PROPERTY PUBLIC fMinCircularity : REFERENCE TO _REAL
GET
fMinCircularity REF= _fMinCircularity;
END_GET
END_PROPERTY

PROPERTY PUBLIC fMinConvexity : REFERENCE TO _REAL
GET
fMinConvexity REF= _fMinConvexity;
END_GET
END_PROPERTY

PROPERTY PUBLIC fMinInertiaRatio : REFERENCE TO _REAL
GET
fMinInertiaRatio REF= _fMinInertiaRatio;
END_GET
END_PROPERTY

PROPERTY PUBLIC fMinThreshold : REFERENCE TO _REAL
GET
fMinThreshold REF= _fMinThreshold;
END_GET
END_PROPERTY

PROPERTY PUBLIC fThresholdStep : REFERENCE TO _REAL
GET
fThresholdStep REF= _fThresholdStep;
END_GET
END_PROPERTY

PROPERTY PUBLIC Identifier : T_MAXSTRING
GET
Identifier := 'TcVnParamsSB';
END_GET
END_PROPERTY

METHOD PUBLIC MakeReferenceTo
VAR_INPUT
	ReferenceTarget : REFERENCE TO TcVnParamsSB;
END_VAR
activeData REF= ReferenceTarget;
SetMemberReference();
END_METHOD

PROPERTY PUBLIC nBlobColor : REFERENCE TO _USINT
GET
nBlobColor REF= _nBlobColor;
END_GET
END_PROPERTY

PROPERTY PUBLIC nMinRepeatability : REFERENCE TO _UDINT
GET
nMinRepeatability REF= _nMinRepeatability;
END_GET
END_PROPERTY

METHOD PROTECTED SetMemberReference
VAR_INPUT
END_VAR
_bFilterByArea.MakeReferenceTo(activeData.bFilterByArea);
_bFilterByCircularity.MakeReferenceTo(activeData.bFilterByCircularity);
_bFilterByColor.MakeReferenceTo(activeData.bFilterByColor);
_bFilterByConvexity.MakeReferenceTo(activeData.bFilterByConvexity);
_bFilterByInertia.MakeReferenceTo(activeData.bFilterByInertia);
_fMinArea.MakeReferenceTo(activeData.fMinArea);
_fMaxArea.MakeReferenceTo(activeData.fMaxArea);
_fMinCircularity.MakeReferenceTo(activeData.fMinCircularity);
_fMaxCircularity.MakeReferenceTo(activeData.fMaxCircularity);
_nBlobColor.MakeReferenceTo(activeData.nBlobColor);
_fMinConvexity.MakeReferenceTo(activeData.fMinConvexity);
_fMaxConvexity.MakeReferenceTo(activeData.fMaxConvexity);
_fMinInertiaRatio.MakeReferenceTo(activeData.fMinInertiaRatio);
_fMaxInertiaRatio.MakeReferenceTo(activeData.fMaxInertiaRatio);
_fMinBlobDist.MakeReferenceTo(activeData.fMinBlobDist);
_nMinRepeatability.MakeReferenceTo(activeData.nMinRepeatability);
_fMinThreshold.MakeReferenceTo(activeData.fMinThreshold);
_fMaxThreshold.MakeReferenceTo(activeData.fMaxThreshold);
_fThresholdStep.MakeReferenceTo(activeData.fThresholdStep);
END_METHOD

PROPERTY PUBLIC Size : UDINT
GET
Size := SIZEOF(activeData);
END_GET
END_PROPERTY

METHOD TryMakeReferenceTo : BOOL
VAR_INPUT
	Target : I_Datatype;
END_VAR
VAR
	pTargetData : POINTER TO TcVnParamsSB;
END_VAR
IF NOT IsEquivalentTo(Target) THEN
	RETURN;
END_IF

pTargetData := Target.Address;
activeData REF= pTargetData^;
SetMemberReference();
TryMakeReferenceTo := TRUE;
END_METHOD

PROPERTY PUBLIC Value : REFERENCE TO TcVnParamsSB
GET
Value REF= activeData;
END_GET
END_PROPERTY

END_FUNCTION_BLOCK

// ---- Datatypes/Structs/_TcVnParamsBRISK.TcPOU
{attribute 'linkalways'} 
{attribute 'no_explicit_call' := 'This FB is a CLASS and must be accessed using methods or properties'}
{attribute 'enable_dynamic_creation'}
FUNCTION_BLOCK _TcVnParamsBRISK EXTENDS StructuredDatatypeBase
VAR
	localData : TcVnParamsBRISK;
	activeData : REFERENCE TO TcVnParamsBRISK REF= localData;
	_nThreshold : _DINT(localData.nThreshold);
	_nOctaves : _UDINT(localData.nOctaves);
	_fPatternScale : _REAL(localData.fPatternScale);
END_VAR

PROPERTY PUBLIC Address : PVOID
GET
Address := ADR(activeData);
END_GET
END_PROPERTY

METHOD PUBLIC ClearReference
VAR_INPUT
END_VAR
activeData REF= localData;
SetMemberReference();
END_METHOD

METHOD PUBLIC Clone : I_Datatype
VAR
    pClone : POINTER TO _TcVnParamsBRISK;
END_VAR
pClone := __NEW(_TcVnParamsBRISK());
pClone^.Value := Value;
Clone := pClone^;
END_METHOD

METHOD FB_init : BOOL
VAR_INPUT
	bInitRetains : BOOL; // if TRUE, the retain variables are initialized (warm start / cold start)
	bInCopyCode : BOOL;  // if TRUE, the instance afterwards gets moved into the copy code (online change)
END_VAR
SetMemberReference();
AddMember('nThreshold', _nThreshold);
AddMember('nOctaves', _nOctaves);
AddMember('fPatternScale', _fPatternScale);
END_METHOD

PROPERTY PUBLIC fPatternScale : REFERENCE TO _REAL
GET
fPatternScale REF= _fPatternScale;
END_GET
END_PROPERTY

PROPERTY PUBLIC Identifier : T_MAXSTRING
GET
Identifier := 'TcVnParamsBRISK';
END_GET
END_PROPERTY

METHOD PUBLIC MakeReferenceTo
VAR_INPUT
	ReferenceTarget : REFERENCE TO TcVnParamsBRISK;
END_VAR
activeData REF= ReferenceTarget;
SetMemberReference();
END_METHOD

PROPERTY PUBLIC nOctaves : REFERENCE TO _UDINT
GET
nOctaves REF= _nOctaves;
END_GET
END_PROPERTY

PROPERTY PUBLIC nThreshold : REFERENCE TO _DINT
GET
nThreshold REF= _nThreshold;
END_GET
END_PROPERTY

METHOD PROTECTED SetMemberReference
VAR_INPUT
END_VAR
_nThreshold.MakeReferenceTo(activeData.nThreshold);
_nOctaves.MakeReferenceTo(activeData.nOctaves);
_fPatternScale.MakeReferenceTo(activeData.fPatternScale);
END_METHOD

PROPERTY PUBLIC Size : UDINT
GET
Size := SIZEOF(activeData);
END_GET
END_PROPERTY

METHOD TryMakeReferenceTo : BOOL
VAR_INPUT
	Target : I_Datatype;
END_VAR
VAR
	pTargetData : POINTER TO TcVnParamsBRISK;
END_VAR
IF NOT IsEquivalentTo(Target) THEN
	RETURN;
END_IF

pTargetData := Target.Address;
activeData REF= pTargetData^;
SetMemberReference();
TryMakeReferenceTo := TRUE;
END_METHOD

PROPERTY PUBLIC Value : REFERENCE TO TcVnParamsBRISK
GET
Value REF= activeData;
END_GET
END_PROPERTY

METHOD PUBLIC TryDeserializeFrom : BOOL
VAR_INPUT
    Deserializer : I_Deserializer;
    Feedback : I_DeserializerFeedback;
END_VAR
VAR
    membersEnumerator : I_DeserializerObjectForwardEnumerator;
    member : I_Datatype;
    memberName : T_MAXSTRING;
END_VAR
// Map the legacy member name without advertising or serializing it twice.
membersEnumerator := Deserializer.GetObjectEnumerator();
WHILE membersEnumerator.MoveNext() DO
    memberName := membersEnumerator.Key;
    IF memberName = 'fPatternScale ' THEN
        memberName := 'fPatternScale';
    END_IF
    IF Members.TryGetMemberByName(memberName, member) THEN
        IF NOT member.TryDeserializeFrom(membersEnumerator.Current, Feedback) THEN
            membersEnumerator.Dispose();
            RETURN;
        END_IF
    END_IF
END_WHILE
membersEnumerator.Dispose();
TryDeserializeFrom := TRUE;
END_METHOD

END_FUNCTION_BLOCK

// ---- Datatypes/Structs/_TcVnParamsFAST.TcPOU
{attribute 'linkalways'} 
{attribute 'no_explicit_call' := 'This FB is a CLASS and must be accessed using methods or properties'}
{attribute 'enable_dynamic_creation'}
FUNCTION_BLOCK _TcVnParamsFAST EXTENDS StructuredDatatypeBase
VAR
	localData : TcVnParamsFAST;
	activeData : REFERENCE TO TcVnParamsFAST REF= localData;
	_nThreshold : _DINT(localData.nThreshold);
    _bNonMaxSuppression : _BOOL(localData.bNonMaxSuppression);
	_eType : _ETcVnKeypointDetectionTypeFAST(localData.eType);
END_VAR

PROPERTY PUBLIC Address : PVOID
GET
Address := ADR(activeData);
END_GET
END_PROPERTY

PROPERTY PUBLIC bNonMaxSuppression : REFERENCE TO _BOOL
GET
bNonMaxSuppression REF= _bNonMaxSuppression;
END_GET
END_PROPERTY

METHOD PUBLIC ClearReference
VAR_INPUT
END_VAR
activeData REF= localData;
SetMemberReference();
END_METHOD

METHOD PUBLIC Clone : I_Datatype
VAR
    pClone : POINTER TO _TcVnParamsFAST;
END_VAR
pClone := __NEW(_TcVnParamsFAST());
pClone^.Value := Value;
Clone := pClone^;
END_METHOD

PROPERTY PUBLIC eType : REFERENCE TO _ETcVnKeypointDetectionTypeFAST
GET
eType REF= _eType;
END_GET
END_PROPERTY

METHOD FB_init : BOOL
VAR_INPUT
	bInitRetains : BOOL; // if TRUE, the retain variables are initialized (warm start / cold start)
	bInCopyCode : BOOL;  // if TRUE, the instance afterwards gets moved into the copy code (online change)
END_VAR
SetMemberReference();
AddMember('nThreshold',_nThreshold);
AddMember('bNonMaxSuppression',_bNonMaxSuppression );
AddMember('eType',_eType);
END_METHOD

PROPERTY PUBLIC Identifier : T_MAXSTRING
GET
Identifier := 'TcVnParamsFAST';
END_GET
END_PROPERTY

METHOD PUBLIC MakeReferenceTo
VAR_INPUT
	ReferenceTarget : REFERENCE TO TcVnParamsFAST;
END_VAR
activeData REF= ReferenceTarget;
SetMemberReference();
END_METHOD

PROPERTY PUBLIC nThreshold : REFERENCE TO _DINT
GET
nThreshold REF= _nThreshold;
END_GET
END_PROPERTY

METHOD PROTECTED SetMemberReference
VAR_INPUT
END_VAR
_nThreshold.MakeReferenceTo(activeData.nThreshold);
_bNonMaxSuppression.MakeReferenceTo(activeData.bNonMaxSuppression);
_eType.MakeReferenceTo(activeData.eType);
END_METHOD

PROPERTY PUBLIC Size : UDINT
GET
Size := SIZEOF(activeData);
END_GET
END_PROPERTY

METHOD TryMakeReferenceTo : BOOL
VAR_INPUT
	Target : I_Datatype;
END_VAR
VAR
	pTargetData : POINTER TO TcVnParamsFAST;
END_VAR
IF NOT IsEquivalentTo(Target) THEN
	RETURN;
END_IF

pTargetData := Target.Address;
activeData REF= pTargetData^;
SetMemberReference();
TryMakeReferenceTo := TRUE;
END_METHOD

PROPERTY PUBLIC Value : REFERENCE TO TcVnParamsFAST
GET
Value REF= activeData;
END_GET
END_PROPERTY

END_FUNCTION_BLOCK

// ---- Datatypes/Structs/_TcVnParamsBlobDetection.TcPOU
{attribute 'linkalways'} 
{attribute 'no_explicit_call' := 'This FB is a CLASS and must be accessed using methods or properties'}
{attribute 'enable_dynamic_creation'}
FUNCTION_BLOCK _TcVnParamsBlobDetection EXTENDS StructuredDatatypeBase
VAR
	localData : TcVnParamsBlobDetection;
	activeData : REFERENCE TO TcVnParamsBlobDetection REF= localData;
    _bFilterByArea         : _BOOL(localdata.bFilterByArea);
    _bFilterByCircularity  : _BOOL(localdata.bFilterByCircularity);
    _bFilterByConvexity    : _BOOL(localdata.bFilterByConvexity);
    _bFilterByEccentricity : _BOOL(localdata.bFilterByEccentricity);
    _bFilterByInertiaRatio : _BOOL(localdata.bFilterByInertiaRatio);
    _fMinArea              : _REAL(localdata.fMinArea);
    _fMaxArea              : _REAL(localdata.fMaxArea);
    _fMinCircularity       : _REAL(localdata.fMinCircularity);
    _fMaxCircularity       : _REAL(localdata.fMaxCircularity);
    _fMinConvexity         : _REAL(localdata.fMinConvexity);
    _fMaxConvexity         : _REAL(localdata.fMaxConvexity);
    _fMinEccentricity      : _REAL(localdata.fMinEccentricity);
    _fMaxEccentricity      : _REAL(localdata.fMaxEccentricity);
    _fMinInertiaRatio      : _REAL(localdata.fMinInertiaRatio);
    _fMaxInertiaRatio      : _REAL(localdata.fMaxInertiaRatio);
    _eThresholdType        : _ETcVnThresholdType(localdata.eThresholdType);
    _fMinThreshold         : _REAL(localdata.fMinThreshold);
    _fMaxThreshold         : _REAL(localdata.fMaxThreshold);
    _fThresholdStep        : _REAL(localdata.fThresholdStep);
    _fMinBlobDistance      : _REAL(localdata.fMinBlobDistance);
    _nMinRepeatability     : _UDINT(localdata.nMinRepeatability);
    _eBlobCombination      : _ETcVnBlobCombination(localdata.eBlobCombination);
    _bExcludeBorderBlobs   : _BOOL(localdata.bExcludeBorderBlobs);
END_VAR

PROPERTY PUBLIC Address : PVOID
GET
Address := ADR(activeData);
END_GET
END_PROPERTY

PROPERTY PUBLIC bExcludeBorderBlobs : REFERENCE TO _BOOL
GET
bExcludeBorderBlobs REF= _bExcludeBorderBlobs;
END_GET
END_PROPERTY

PROPERTY PUBLIC bFilterByArea : REFERENCE TO _BOOL
GET
bFilterByArea REF= _bFilterByArea;
END_GET
END_PROPERTY

PROPERTY PUBLIC bFilterByCircularity : REFERENCE TO _BOOL
GET
bFilterByCircularity REF= _bFilterByCircularity;
END_GET
END_PROPERTY

PROPERTY PUBLIC bFilterByConvexity : REFERENCE TO _BOOL
GET
bFilterByConvexity REF= _bFilterByConvexity;
END_GET
END_PROPERTY

PROPERTY PUBLIC bFilterByEccentricity : REFERENCE TO _BOOL
GET
bFilterByEccentricity REF= _bFilterByEccentricity;
END_GET
END_PROPERTY

PROPERTY PUBLIC bFilterByInertiaRatio : REFERENCE TO _BOOL
GET
bFilterByInertiaRatio REF= _bFilterByInertiaRatio;
END_GET
END_PROPERTY

METHOD PUBLIC ClearReference
VAR_INPUT
END_VAR
activeData REF= localData;
SetMemberReference();
END_METHOD

METHOD PUBLIC Clone : I_Datatype
VAR
    pClone : POINTER TO _TcVnParamsBlobDetection;
END_VAR
pClone := __NEW(_TcVnParamsBlobDetection());
pClone^.Value := Value;
Clone := pClone^;
END_METHOD

PROPERTY PUBLIC eBlobCombination : REFERENCE TO _ETcVnBlobCombination
GET
eBlobCombination REF= _eBlobCombination;
END_GET
END_PROPERTY

PROPERTY PUBLIC eThresholdType : REFERENCE TO _ETcVnThresholdType
GET
eThresholdType REF= _eThresholdType;
END_GET
END_PROPERTY

METHOD FB_init : BOOL
VAR_INPUT
	bInitRetains : BOOL; // if TRUE, the retain variables are initialized (warm start / cold start)
	bInCopyCode : BOOL;  // if TRUE, the instance afterwards gets moved into the copy code (online change)
END_VAR
SetMemberReference();
AddMember('bFilterByArea', _bFilterByArea);
AddMember('bFilterByCircularity', _bFilterByCircularity);
AddMember('bFilterByConvexity', _bFilterByConvexity);
AddMember('bFilterByEccentricity', _bFilterByEccentricity);
AddMember('bFilterByInertiaRatio', _bFilterByInertiaRatio);
AddMember('fMinArea', _fMinArea);
AddMember('fMaxArea', _fMaxArea);
AddMember('fMinCircularity', _fMinCircularity);
AddMember('fMaxCircularity', _fMaxCircularity);
AddMember('fMinConvexity', _fMinConvexity);
AddMember('fMaxConvexity', _fMaxConvexity);
AddMember('fMinEccentricity', _fMinEccentricity);
AddMember('fMaxEccentricity', _fMaxEccentricity);
AddMember('fMinInertiaRatio', _fMinInertiaRatio);
AddMember('fMaxInertiaRatio', _fMaxInertiaRatio);
AddMember('eThresholdType', _eThresholdType);
AddMember('fMinThreshold', _fMinThreshold);
AddMember('fMaxThreshold', _fMaxThreshold);
AddMember('fThresholdStep',  _fThresholdStep);
AddMember('fMinBlobDistance', _fMinBlobDistance);
AddMember('nMinRepeatability', _nMinRepeatability);
AddMember('eBlobCombination', _eBlobCombination);
AddMember('bExcludeBorderBlobs', _bExcludeBorderBlobs);
END_METHOD

PROPERTY PUBLIC fMaxArea : REFERENCE TO _REAL
GET
fMaxArea REF= _fMaxArea;
END_GET
END_PROPERTY

PROPERTY PUBLIC fMaxCircularity : REFERENCE TO _REAL
GET
fMaxCircularity REF= _fMaxCircularity;
END_GET
END_PROPERTY

PROPERTY PUBLIC fMaxConvexity : REFERENCE TO _REAL
GET
fMaxConvexity REF= _fMaxConvexity;
END_GET
END_PROPERTY

PROPERTY PUBLIC fMaxEccentricity : REFERENCE TO _REAL
GET
fMaxEccentricity REF= _fMaxEccentricity;
END_GET
END_PROPERTY

PROPERTY PUBLIC fMaxInertiaRatio : REFERENCE TO _REAL
GET
fMaxInertiaRatio REF= _fMaxInertiaRatio;
END_GET
END_PROPERTY

PROPERTY PUBLIC fMaxThreshold : REFERENCE TO _REAL
GET
fMaxThreshold REF= _fMaxThreshold;
END_GET
END_PROPERTY

PROPERTY PUBLIC fMinArea : REFERENCE TO _REAL
GET
fMinArea REF= _fMinArea;
END_GET
END_PROPERTY

PROPERTY PUBLIC fMinBlobDistance : REFERENCE TO _REAL
GET
fMinBlobDistance REF= _fMinBlobDistance;
END_GET
END_PROPERTY

PROPERTY PUBLIC fMinCircularity : REFERENCE TO _REAL
GET
fMinCircularity REF= _fMinCircularity;
END_GET
END_PROPERTY

PROPERTY PUBLIC fMinConvexity : REFERENCE TO _REAL
GET
fMinConvexity REF= _fMinConvexity;
END_GET
END_PROPERTY

PROPERTY PUBLIC fMinEccentricity : REFERENCE TO _REAL
GET
fMinEccentricity REF= _fMinEccentricity;
END_GET
END_PROPERTY

PROPERTY PUBLIC fMinInertiaRatio : REFERENCE TO _REAL
GET
fMinInertiaRatio REF= _fMinInertiaRatio;
END_GET
END_PROPERTY

PROPERTY PUBLIC fMinThreshold : REFERENCE TO _REAL
GET
fMinThreshold REF= _fMinThreshold;
END_GET
END_PROPERTY

PROPERTY PUBLIC fThresholdStep : REFERENCE TO _REAL
GET
fThresholdStep REF= _fThresholdStep;
END_GET
END_PROPERTY

PROPERTY PUBLIC Identifier : T_MAXSTRING
GET
Identifier := 'TcVnParamsBlobDetection';
END_GET
END_PROPERTY

METHOD PUBLIC MakeReferenceTo
VAR_INPUT
	ReferenceTarget : REFERENCE TO TcVnParamsBlobDetection;
END_VAR
activeData REF= ReferenceTarget;
SetMemberReference();
END_METHOD

PROPERTY PUBLIC nMinRepeatability : REFERENCE TO _UDINT
GET
nMinRepeatability REF= _nMinRepeatability;
END_GET
END_PROPERTY

METHOD PROTECTED SetMemberReference
VAR_INPUT
END_VAR
_bFilterByArea.MakeReferenceTo(activeData.bFilterByArea);
_bFilterByCircularity.MakeReferenceTo(activeData.bFilterByCircularity);
_bFilterByConvexity.MakeReferenceTo(activeData.bFilterByConvexity);
_bFilterByEccentricity.MakeReferenceTo(activeData.bFilterByEccentricity);
_bFilterByInertiaRatio.MakeReferenceTo(activeData.bFilterByInertiaRatio);
_fMinArea.MakeReferenceTo(activeData.fMinArea);
_fMaxArea.MakeReferenceTo(activeData.fMaxArea);
_fMinCircularity.MakeReferenceTo(activeData.fMinCircularity);
_fMaxCircularity.MakeReferenceTo(activeData.fMaxCircularity);
_fMinConvexity.MakeReferenceTo(activeData.fMinConvexity);
_fMaxConvexity.MakeReferenceTo(activeData.fMaxConvexity);
_fMinEccentricity.MakeReferenceTo(activeData.fMinEccentricity);
_fMaxEccentricity.MakeReferenceTo(activeData.fMaxEccentricity);
_fMinInertiaRatio.MakeReferenceTo(activeData.fMinInertiaRatio);
_fMaxInertiaRatio.MakeReferenceTo(activeData.fMaxInertiaRatio);
_eThresholdType.MakeReferenceTo(activeData.eThresholdType);
_fMinThreshold.MakeReferenceTo(activeData.fMinThreshold);
_fMaxThreshold.MakeReferenceTo(activeData.fMaxThreshold);
_fThresholdStep.MakeReferenceTo(activeData.fThresholdStep);
_fMinBlobDistance.MakeReferenceTo(activeData.fMinBlobDistance);
_nMinRepeatability.MakeReferenceTo(activeData.nMinRepeatability);
_eBlobCombination.MakeReferenceTo(activeData.eBlobCombination);
_bExcludeBorderBlobs.MakeReferenceTo(activeData.bExcludeBorderBlobs);
END_METHOD

PROPERTY PUBLIC Size : UDINT
GET
Size := SIZEOF(activeData);
END_GET
END_PROPERTY

METHOD TryMakeReferenceTo : BOOL
VAR_INPUT
	Target : I_Datatype;
END_VAR
VAR
	pTargetData : POINTER TO TcVnParamsBlobDetection;
END_VAR
IF NOT IsEquivalentTo(Target) THEN
	RETURN;
END_IF

pTargetData := Target.Address;
activeData REF= pTargetData^;
SetMemberReference();
TryMakeReferenceTo := TRUE;
END_METHOD

PROPERTY PUBLIC Value : REFERENCE TO TcVnParamsBlobDetection
GET
Value REF= activeData;
END_GET
END_PROPERTY

END_FUNCTION_BLOCK

// ---- Datatypes/Structs/_TcVnCameraCalibrationOptions.TcPOU
{attribute 'linkalways'} 
{attribute 'no_explicit_call' := 'This FB is a CLASS and must be accessed using methods or properties'}
{attribute 'enable_dynamic_creation'}
FUNCTION_BLOCK _TcVnCameraCalibrationOptions EXTENDS StructuredDatatypeBase
VAR
	localData : TcVnCameraCalibrationOptions;
	activeData : REFERENCE TO TcVnCameraCalibrationOptions REF= localData;

    _bUseIntrinsicGuess : _BIT();
    _bFixAspectRatio    : _BIT();
    _bFixPrincipalPoint : _BIT();
    _bZeroTangentDist   : _BIT();
    _bFixFocalLength    : _BIT();
    _bFixK1             : _BIT();
    _bFixK2             : _BIT();
    _bFixK3             : _BIT();
    _bFixK4             : _BIT();
    _bFixK5             : _BIT();
    _bFixK6             : _BIT();
    _bRationalModel     : _BIT();
END_VAR

PROPERTY PUBLIC Address : PVOID
GET
Address := ADR(activeData);
END_GET
END_PROPERTY

PROPERTY PUBLIC bFixAspectRatio : REFERENCE TO _BIT
GET
bFixAspectRatio REF= _bFixAspectRatio;
END_GET
END_PROPERTY

PROPERTY PUBLIC bFixFocalLength : REFERENCE TO _BIT
GET
bFixFocalLength REF= _bFixFocalLength;
END_GET
END_PROPERTY

PROPERTY PUBLIC bFixK1 : REFERENCE TO _BIT
GET
bFixK1 REF= _bFixK1;
END_GET
END_PROPERTY

PROPERTY PUBLIC bFixK2 : REFERENCE TO _BIT
GET
bFixK2 REF= _bFixK2;
END_GET
END_PROPERTY

PROPERTY PUBLIC bFixK3 : REFERENCE TO _BIT
GET
bFixK3 REF= _bFixK3;
END_GET
END_PROPERTY

PROPERTY PUBLIC bFixK4 : REFERENCE TO _BIT
GET
bFixK4 REF= _bFixK4;
END_GET
END_PROPERTY

PROPERTY PUBLIC bFixK5 : REFERENCE TO _BIT
GET
bFixK5 REF= _bFixK5;
END_GET
END_PROPERTY

PROPERTY PUBLIC bFixK6 : REFERENCE TO _BIT
GET
bFixK6 REF= _bFixK6;
END_GET
END_PROPERTY

PROPERTY PUBLIC bFixPrincipalPoint : REFERENCE TO _BIT
GET
bFixPrincipalPoint REF= _bFixPrincipalPoint;
END_GET
END_PROPERTY

PROPERTY PUBLIC bRationalModel : REFERENCE TO _BIT
GET
bRationalModel REF= _bRationalModel;
END_GET
END_PROPERTY

PROPERTY PUBLIC bUseIntrinsicGuess : REFERENCE TO _BIT
GET
bUseIntrinsicGuess REF= _bUseIntrinsicGuess;
END_GET
END_PROPERTY

PROPERTY PUBLIC bZeroTangentDist : REFERENCE TO _BIT
GET
bZeroTangentDist REF= _bZeroTangentDist;
END_GET
END_PROPERTY

METHOD PUBLIC ClearReference
VAR_INPUT
END_VAR
activeData REF= localData;
SetMemberReference();
END_METHOD

METHOD PUBLIC Clone : I_Datatype
VAR
    pClone : POINTER TO _TcVnCameraCalibrationOptions;
END_VAR
pClone := __NEW(_TcVnCameraCalibrationOptions());
pClone^.Value := Value;
Clone := pClone^;
END_METHOD

METHOD FB_init : BOOL
VAR_INPUT
	bInitRetains : BOOL; // if TRUE, the retain variables are initialized (warm start / cold start)
	bInCopyCode : BOOL;  // if TRUE, the instance afterwards gets moved into the copy code (online change)
END_VAR
SetMemberReference();
AddMember('bUseIntrinsicGuess',_bUseIntrinsicGuess);
AddMember('bFixAspectRatio',_bFixAspectRatio);
AddMember('bFixPrincipalPoint',_bFixPrincipalPoint);
AddMember('bZeroTangentDist',_bZeroTangentDist);
AddMember('bFixFocalLength',_bFixFocalLength);
AddMember('bFixK1',_bFixK1);
AddMember('bFixK2',_bFixK2);
AddMember('bFixK3',_bFixK3);
AddMember('bFixK4',_bFixK4);
AddMember('bFixK5',_bFixK5);
AddMember('bFixK6',_bFixK6);
AddMember('bRationalModel',_bRationalModel);
END_METHOD

PROPERTY PUBLIC Identifier : T_MAXSTRING
GET
Identifier := 'TcVnCameraCalibrationOptions';
END_GET
END_PROPERTY

METHOD PUBLIC MakeReferenceTo
VAR_INPUT
	ReferenceTarget : REFERENCE TO TcVnCameraCalibrationOptions;
END_VAR
activeData REF= ReferenceTarget;
SetMemberReference();
END_METHOD

METHOD PROTECTED SetMemberReference
VAR_STAT
	// this variable is used for BITADR as this function fails if used on a local variable.
	structure : TcVnCameraCalibrationOptions;
END_VAR
_bUseIntrinsicGuess.MakeReferenceTo(THIS^, GetByteOffset(localData, localData.bUseIntrinsicGuess), BITADR(structure.bUseIntrinsicGuess));
_bFixAspectRatio.MakeReferenceTo(THIS^, GetByteOffset(localData, localData.bFixAspectRatio), BITADR(structure.bFixAspectRatio));
_bFixPrincipalPoint.MakeReferenceTo(THIS^, GetByteOffset(localData, localData.bFixPrincipalPoint), BITADR(structure.bFixPrincipalPoint));
_bZeroTangentDist.MakeReferenceTo(THIS^, GetByteOffset(localData, localData.bZeroTangentDist), BITADR(structure.bZeroTangentDist));
_bFixFocalLength.MakeReferenceTo(THIS^, GetByteOffset(localData, localData.bFixFocalLength), BITADR(structure.bFixFocalLength));
_bFixK1.MakeReferenceTo(THIS^, GetByteOffset(localData, localData.bFixK1), BITADR(structure.bFixK1));
_bFixK2.MakeReferenceTo(THIS^, GetByteOffset(localData, localData.bFixK2), BITADR(structure.bFixK2));
_bFixK3.MakeReferenceTo(THIS^, GetByteOffset(localData, localData.bFixK3), BITADR(structure.bFixK3));
_bFixK4.MakeReferenceTo(THIS^, GetByteOffset(localData, localData.bFixK4), BITADR(structure.bFixK4));
_bFixK5.MakeReferenceTo(THIS^, GetByteOffset(localData, localData.bFixK5), BITADR(structure.bFixK5));
_bFixK6.MakeReferenceTo(THIS^, GetByteOffset(localData, localData.bFixK6), BITADR(structure.bFixK6));
_bRationalModel.MakeReferenceTo(THIS^, GetByteOffset(localData, localData.bRationalModel), BITADR(structure.bRationalModel));
END_METHOD

PROPERTY PUBLIC Size : UDINT
GET
Size := SIZEOF(activeData);
END_GET
END_PROPERTY

METHOD TryMakeReferenceTo : BOOL
VAR_INPUT
	Target : I_Datatype;
END_VAR
VAR
	pTargetData : POINTER TO TcVnCameraCalibrationOptions;
END_VAR
IF NOT IsEquivalentTo(Target) THEN
	RETURN;
END_IF

pTargetData := Target.Address;
activeData REF= pTargetData^;
SetMemberReference();
TryMakeReferenceTo := TRUE;
END_METHOD

PROPERTY PUBLIC Value : REFERENCE TO TcVnCameraCalibrationOptions
GET
Value REF= activeData;
END_GET
END_PROPERTY

END_FUNCTION_BLOCK

// ---- Datatypes/Structs/_TcVnParamsGFTT.TcPOU
{attribute 'linkalways'} 
{attribute 'no_explicit_call' := 'This FB is a CLASS and must be accessed using methods or properties'}
{attribute 'enable_dynamic_creation'}
FUNCTION_BLOCK _TcVnParamsGFTT EXTENDS StructuredDatatypeBase
VAR
	localData : TcVnParamsGFTT;
	activeData : REFERENCE TO TcVnParamsGFTT REF= localData;
	_nMaxCorners : _UDINT(localData.nMaxCorners);
    _fQualityLevel : _LREAL(localData.fQualityLevel);
	_fMinDistance : _LREAL(localData.fMinDistance);
	_nBlockSize : _UDINT(localData.nBlockSize);
	_bUseHarrisDetector : _BOOL(localData.bUseHarrisDetector);
	_fHarrisK : _LREAL(localData.fHarrisK);
END_VAR

PROPERTY PUBLIC Address : PVOID
GET
Address := ADR(activeData);
END_GET
END_PROPERTY

PROPERTY PUBLIC bUseHarrisDetector : REFERENCE TO _BOOL
GET
bUseHarrisDetector REF= _bUseHarrisDetector;
END_GET
END_PROPERTY

METHOD PUBLIC ClearReference
VAR_INPUT
END_VAR
activeData REF= localData;
SetMemberReference();
END_METHOD

METHOD PUBLIC Clone : I_Datatype
VAR
    pClone : POINTER TO _TcVnParamsGFTT;
END_VAR
pClone := __NEW(_TcVnParamsGFTT());
pClone^.Value := Value;
Clone := pClone^;
END_METHOD

METHOD FB_init : BOOL
VAR_INPUT
	bInitRetains : BOOL; // if TRUE, the retain variables are initialized (warm start / cold start)
	bInCopyCode : BOOL;  // if TRUE, the instance afterwards gets moved into the copy code (online change)
END_VAR
SetMemberReference();
AddMember('nMaxCorners', _nMaxCorners);
AddMember('fQualityLevel', _fQualityLevel);
AddMember('fMinDistance', _fMinDistance);
AddMember('nBlockSize', _nBlockSize);
AddMember('bUseHarrisDetector', _bUseHarrisDetector);
AddMember('fHarrisK', _fHarrisK);
END_METHOD

PROPERTY PUBLIC fHarrisK : REFERENCE TO _LREAL
GET
fHarrisK REF= _fHarrisK;
END_GET
END_PROPERTY

PROPERTY PUBLIC fMinDistance : REFERENCE TO _LREAL
GET
fMinDistance REF= _fMinDistance;
END_GET
END_PROPERTY

PROPERTY PUBLIC fQualityLevel : REFERENCE TO _LREAL
GET
fQualityLevel REF= _fQualityLevel;
END_GET
END_PROPERTY

PROPERTY PUBLIC Identifier : T_MAXSTRING
GET
Identifier := 'TcVnParamsGFTT';
END_GET
END_PROPERTY

METHOD PUBLIC MakeReferenceTo
VAR_INPUT
	ReferenceTarget : REFERENCE TO TcVnParamsGFTT;
END_VAR
activeData REF= ReferenceTarget;
SetMemberReference();
END_METHOD

PROPERTY PUBLIC nBlockSize : REFERENCE TO _UDINT
GET
nBlockSize REF= _nBlockSize;
END_GET
END_PROPERTY

PROPERTY PUBLIC nMaxCorners : REFERENCE TO _UDINT
GET
nMaxCorners REF= _nMaxCorners;
END_GET
END_PROPERTY

METHOD PROTECTED SetMemberReference
VAR_INPUT
END_VAR
_nMaxCorners.MakeReferenceTo(activeData.nMaxCorners);
_fQualityLevel.MakeReferenceTo(activeData.fQualityLevel);
_fMinDistance.MakeReferenceTo(activeData.fMinDistance);
_nBlockSize.MakeReferenceTo(activeData.nBlockSize);
_bUseHarrisDetector.MakeReferenceTo(activeData.bUseHarrisDetector);
_fHarrisK.MakeReferenceTo(activeData.fHarrisK);
END_METHOD

PROPERTY PUBLIC Size : UDINT
GET
Size := SIZEOF(activeData);
END_GET
END_PROPERTY

METHOD TryMakeReferenceTo : BOOL
VAR_INPUT
	Target : I_Datatype;
END_VAR
VAR
	pTargetData : POINTER TO TcVnParamsGFTT;
END_VAR
IF NOT IsEquivalentTo(Target) THEN
	RETURN;
END_IF

pTargetData := Target.Address;
activeData REF= pTargetData^;
SetMemberReference();
TryMakeReferenceTo := TRUE;
END_METHOD

PROPERTY PUBLIC Value : REFERENCE TO TcVnParamsGFTT
GET
Value REF= activeData;
END_GET
END_PROPERTY

END_FUNCTION_BLOCK

// ---- Datatypes/Structs/_TcVnRotatedRectangle.TcPOU
{attribute 'linkalways'} 
{attribute 'no_explicit_call' := 'This FB is a CLASS and must be accessed using methods or properties'}
{attribute 'enable_dynamic_creation'}
FUNCTION_BLOCK _TcVnRotatedRectangle EXTENDS StructuredDatatypeBase
VAR
	localData : TcVnRotatedRectangle;
	activeData : REFERENCE TO TcVnRotatedRectangle REF= localData;
    _aCenter : _TcVnPoint2_REAL();
    _stSize : _TcVnSize2_REAL();
    _fAngle : _REAL(localdata.fAngle);
END_VAR

PROPERTY PUBLIC aCenter : REFERENCE TO _TcVnPoint2_REAL
GET
aCenter REF= _aCenter;
END_GET
END_PROPERTY

PROPERTY PUBLIC Address : PVOID
GET
Address := ADR(activeData);
END_GET
END_PROPERTY

METHOD PUBLIC ClearReference
VAR_INPUT
END_VAR
activeData REF= localData;
SetMemberReference();
END_METHOD

METHOD PUBLIC Clone : I_Datatype
VAR
    pClone : POINTER TO _TcVnRotatedRectangle;
END_VAR
pClone := __NEW(_TcVnRotatedRectangle());
pClone^.Value := Value;
Clone := pClone^;
END_METHOD

PROPERTY PUBLIC fAngle : REFERENCE TO _REAL
GET
fAngle REF= _fAngle;
END_GET
END_PROPERTY

METHOD FB_init : BOOL
VAR_INPUT
	bInitRetains : BOOL; // if TRUE, the retain variables are initialized (warm start / cold start)
	bInCopyCode : BOOL;  // if TRUE, the instance afterwards gets moved into the copy code (online change)
END_VAR
SetMemberReference();
AddMember('aCenter', _aCenter);
AddMember('stSize', _stSize);
AddMember('fAngle', _fAngle);
END_METHOD

PROPERTY PUBLIC Identifier : T_MAXSTRING
GET
Identifier := 'TcVnRotatedRectangle';
END_GET
END_PROPERTY

METHOD PUBLIC MakeReferenceTo
VAR_INPUT
	ReferenceTarget : REFERENCE TO TcVnRotatedRectangle;
END_VAR
activeData REF= ReferenceTarget;
SetMemberReference();
END_METHOD

METHOD PROTECTED SetMemberReference
VAR_INPUT
END_VAR
_aCenter.MakeReferenceTo(activeData.aCenter);
_stsize.MakeReferenceTo(activeData.stSize);
_fAngle.MakeReferenceTo(activeData.fAngle);
END_METHOD

PROPERTY PUBLIC Size : UDINT
GET
Size := SIZEOF(activeData);
END_GET
END_PROPERTY

PROPERTY PUBLIC stSize : REFERENCE TO _TcVnSize2_REAL
GET
stSize REF= _stSize;
END_GET
END_PROPERTY

METHOD TryMakeReferenceTo : BOOL
VAR_INPUT
	Target : I_Datatype;
END_VAR
VAR
	pTargetData : POINTER TO TcVnRotatedRectangle;
END_VAR
IF NOT IsEquivalentTo(Target) THEN
	RETURN;
END_IF

pTargetData := Target.Address;
activeData REF= pTargetData^;
SetMemberReference();
TryMakeReferenceTo := TRUE;
END_METHOD

PROPERTY PUBLIC Value : REFERENCE TO TcVnRotatedRectangle
GET
Value REF= activeData;
END_GET
END_PROPERTY

END_FUNCTION_BLOCK

// ---- Datatypes/Structs/_TcVnCircularArc.TcPOU
{attribute 'linkalways'} 
{attribute 'no_explicit_call' := 'This FB is a CLASS and must be accessed using methods or properties'}
{attribute 'enable_dynamic_creation'}
FUNCTION_BLOCK _TcVnCircularArc EXTENDS StructuredDatatypeBase
VAR
	localData : TcVnCircularArc;
	activeData : REFERENCE TO TcVnCircularArc REF= localData;
    _aCenter : _TcVnPoint2_REAL();
    _fRadius : _REAL(localdata.fRadius);
    _fStartAngle : _REAL(localdata.fStartAngle);
    _fEndAngle : _REAL(localdata.fEndAngle);
END_VAR

PROPERTY PUBLIC aCenter : REFERENCE TO _TcVnPoint2_REAL
GET
aCenter REF= _aCenter;
END_GET
END_PROPERTY

PROPERTY PUBLIC Address : PVOID
GET
Address := ADR(activeData);
END_GET
END_PROPERTY

METHOD PUBLIC ClearReference
VAR_INPUT
END_VAR
activeData REF= localData;
SetMemberReference();
END_METHOD

METHOD PUBLIC Clone : I_Datatype
VAR
    pClone : POINTER TO _TcVnCircularArc;
END_VAR
pClone := __NEW(_TcVnCircularArc());
pClone^.Value := Value;
Clone := pClone^;
END_METHOD

METHOD FB_init : BOOL
VAR_INPUT
	bInitRetains : BOOL; // if TRUE, the retain variables are initialized (warm start / cold start)
	bInCopyCode : BOOL;  // if TRUE, the instance afterwards gets moved into the copy code (online change)
END_VAR
SetMemberReference();
AddMember('aCenter', _aCenter);
AddMember('fRadius', _fRadius);
AddMember('fStartAngle', _fStartAngle);
AddMember('fEndAngle', _fEndAngle);
END_METHOD

PROPERTY PUBLIC fEndAngle : REFERENCE TO _REAL
GET
fEndAngle REF= _fEndAngle;
END_GET
END_PROPERTY

PROPERTY PUBLIC fRadius : REFERENCE TO _REAL
GET
fRadius REF= _fRadius;
END_GET
END_PROPERTY

PROPERTY PUBLIC fStartAngle : REFERENCE TO _REAL
GET
fStartAngle REF= _fStartAngle;
END_GET
END_PROPERTY

PROPERTY PUBLIC Identifier : T_MAXSTRING
GET
Identifier := 'TcVnCircularArc';
END_GET
END_PROPERTY

METHOD PUBLIC MakeReferenceTo
VAR_INPUT
	ReferenceTarget : REFERENCE TO TcVnCircularArc;
END_VAR
activeData REF= ReferenceTarget;
SetMemberReference();
END_METHOD

METHOD PROTECTED SetMemberReference
VAR_INPUT
END_VAR
_aCenter.MakeReferenceTo(activeData.aCenter);
_fRadius.MakeReferenceTo(activeData.fRadius);
_fStartAngle.MakeReferenceTo(activeData.fStartAngle);
_fEndAngle.MakeReferenceTo(activeData.fEndAngle);
END_METHOD

PROPERTY PUBLIC Size : UDINT
GET
Size := SIZEOF(activeData);
END_GET
END_PROPERTY

METHOD TryMakeReferenceTo : BOOL
VAR_INPUT
	Target : I_Datatype;
END_VAR
VAR
	pTargetData : POINTER TO TcVnCircularArc;
END_VAR
IF NOT IsEquivalentTo(Target) THEN
	RETURN;
END_IF

pTargetData := Target.Address;
activeData REF= pTargetData^;
SetMemberReference();
TryMakeReferenceTo := TRUE;
END_METHOD

PROPERTY PUBLIC Value : REFERENCE TO TcVnCircularArc
GET
Value REF= activeData;
END_GET
END_PROPERTY

END_FUNCTION_BLOCK

// ---- Datatypes/Structs/_TcVnPixelFormat.TcPOU
{attribute 'linkalways'} 
{attribute 'no_explicit_call' := 'This FB is a CLASS and must be accessed using methods or properties'}
{attribute 'enable_dynamic_creation'}
FUNCTION_BLOCK _TcVnPixelFormat EXTENDS StructuredDatatypeBase
VAR
	localData : TcVnPixelFormat;
	activeData : REFERENCE TO TcVnPixelFormat REF= localData;

	_bSupported : _BIT();
	_bSigned : _BIT();
	_bPlanar : _BIT();
	_bFloat : _BIT();
	_nChannels : _BYTE(localData.nChannels);
	_ePixelEncoding : _ETcVnPixelEncoding(localData.ePixelEncoding);
	_ePixelPackMode : _ETcVnPixelPackMode(localData.ePixelPackMode);
	_nElementSize : _UINT(localData.nElementSize);
	_nTotalSize : _UINT(localData.nTotalSize);
END_VAR

PROPERTY PUBLIC Address : PVOID
GET
Address := ADR(activeData);
END_GET
END_PROPERTY

PROPERTY PUBLIC bFloat : Reference to _BIT
GET
bFloat REF= _bFloat;
END_GET
END_PROPERTY

PROPERTY PUBLIC bPlanar : Reference to _BIT
GET
bPlanar REF= _bPlanar;
END_GET
END_PROPERTY

PROPERTY PUBLIC bSigned : Reference to _BIT
GET
bSigned REF= _bSigned;
END_GET
END_PROPERTY

PROPERTY PUBLIC bSupported : Reference to _BIT
GET
bSupported REF= _bSupported;
END_GET
END_PROPERTY

METHOD PUBLIC ClearReference
VAR_INPUT
END_VAR
activeData REF= localData;
SetMemberReference();
END_METHOD

METHOD PUBLIC Clone : I_Datatype
VAR
    pClone : POINTER TO _TcVnPixelFormat;
END_VAR
pClone := __NEW(_TcVnPixelFormat());
pClone^.Value := Value;
Clone := pClone^;
END_METHOD

PROPERTY PUBLIC ePixelEncoding : Reference to _ETcVnPixelEncoding
GET
ePixelEncoding REF= _ePixelEncoding;
END_GET
END_PROPERTY

PROPERTY PUBLIC ePixelPackMode : Reference to _ETcVnPixelPackMode
GET
ePixelPackMode REF= _ePixelPackMode;
END_GET
END_PROPERTY

METHOD FB_init : BOOL
VAR_INPUT
	bInitRetains : BOOL; // if TRUE, the retain variables are initialized (warm start / cold start)
	bInCopyCode : BOOL;  // if TRUE, the instance afterwards gets moved into the copy code (online change)
END_VAR
SetMemberReference();
AddMember('bSupported',_bSupported);
AddMember('bSigned',_bSigned);
AddMember('bPlanar',_bPlanar);
AddMember('bFloat',_bFloat);
AddMember('nChannels',_nChannels);
AddMember('ePixelEncoding',_ePixelEncoding);
AddMember('ePixelPackMode',_ePixelPackMode);
AddMember('nElementSize',_nElementSize);
AddMember('nTotalSize',_nTotalSize);
END_METHOD

PROPERTY PUBLIC Identifier : T_MAXSTRING
GET
Identifier := 'TcVnPixelFormat';
END_GET
END_PROPERTY

METHOD PUBLIC MakeReferenceTo
VAR_INPUT
	ReferenceTarget : REFERENCE TO TcVnPixelFormat;
END_VAR
activeData REF= ReferenceTarget;
SetMemberReference();
END_METHOD

PROPERTY PUBLIC nChannels : Reference to _BYTE
GET
nChannels REF= _nChannels;
END_GET
END_PROPERTY

PROPERTY PUBLIC nElementSize : Reference to _UINT
GET
nElementSize REF= _nElementSize;
END_GET
END_PROPERTY

PROPERTY PUBLIC nTotalSize : Reference to _UINT
GET
nTotalSize REF= _nTotalSize;
END_GET
END_PROPERTY

METHOD PROTECTED SetMemberReference
VAR_STAT
	// this variable is used for BITADR as this function fails if used on a local variable.
	structure : TcVnPixelFormat;
END_VAR
_bSupported.MakeReferenceTo(THIS^, GetByteOffset(localData, localData.bSupported), BITADR(structure.bSupported));
_bSigned.MakeReferenceTo(THIS^, GetByteOffset(localData, localData.bSigned), BITADR(structure.bSigned));
_bPlanar.MakeReferenceTo(THIS^, GetByteOffset(localData, localData.bPlanar), BITADR(structure.bPlanar));
_bFloat.MakeReferenceTo(THIS^, GetByteOffset(localData, localData.bFloat), BITADR(structure.bFloat));
_nChannels.MakeReferenceTo(activeData.nChannels);
_ePixelEncoding.MakeReferenceTo(activeData.ePixelEncoding);
_ePixelPackMode.MakeReferenceTo(activeData.ePixelPackMode);
_nElementSize.MakeReferenceTo(activeData.nElementSize);
_nTotalSize.MakeReferenceTo(activeData.nTotalSize);
END_METHOD

PROPERTY PUBLIC Size : UDINT
GET
Size := SIZEOF(activeData);
END_GET
END_PROPERTY

METHOD TryMakeReferenceTo : BOOL
VAR_INPUT
	Target : I_Datatype;
END_VAR
VAR
	pTargetData : POINTER TO TcVnPixelFormat;
END_VAR
IF NOT IsEquivalentTo(Target) THEN
	RETURN;
END_IF

pTargetData := Target.Address;
activeData REF= pTargetData^;
SetMemberReference();
TryMakeReferenceTo := TRUE;
END_METHOD

PROPERTY PUBLIC Value : reference to TcVnPixelFormat
GET
Value REF= activeData;
END_GET
END_PROPERTY

END_FUNCTION_BLOCK

// ---- Datatypes/Structs/_TcVnRectangle_DINT.TcPOU
{attribute 'linkalways'} 
{attribute 'no_explicit_call' := 'This FB is a CLASS and must be accessed using methods or properties'}
{attribute 'enable_dynamic_creation'}
FUNCTION_BLOCK _TcVnRectangle_DINT EXTENDS StructuredDatatypeBase
VAR
	localData : TcVnRectangle_DINT;
	activeData : REFERENCE TO TcVnRectangle_DINT REF= localData;
	_nX : _DINT(localData.nX);
	_nY : _DINT(localData.nY);
    _nWidth : _DINT(localData.nWidth);
	_nHeight : _DINT(localData.nHeight);
END_VAR

PROPERTY PUBLIC Address : PVOID
GET
Address := ADR(activeData);
END_GET
END_PROPERTY

METHOD PUBLIC ClearReference
VAR_INPUT
END_VAR
activeData REF= localData;
SetMemberReference();
END_METHOD

METHOD PUBLIC Clone : I_Datatype
VAR
    pClone : POINTER TO _TcVnRectangle_DINT;
END_VAR
pClone := __NEW(_TcVnRectangle_DINT());
pClone^.Value := Value;
Clone := pClone^;
END_METHOD

METHOD FB_init : BOOL
VAR_INPUT
	bInitRetains : BOOL; // if TRUE, the retain variables are initialized (warm start / cold start)
	bInCopyCode : BOOL;  // if TRUE, the instance afterwards gets moved into the copy code (online change)
END_VAR
SetMemberReference();
AddMember('nX',_nX);
AddMember('nY',_nY);
AddMember('nWidth',_nWidth);
AddMember('nHeight',_nHeight);
END_METHOD

PROPERTY PUBLIC Identifier : T_MAXSTRING
GET
Identifier := 'TcVnRectangle_DINT';
END_GET
END_PROPERTY

METHOD PUBLIC MakeReferenceTo
VAR_INPUT
	ReferenceTarget : REFERENCE TO TcVnRectangle_DINT;
END_VAR
activeData REF= ReferenceTarget;
SetMemberReference();
END_METHOD

PROPERTY PUBLIC nHeight : REFERENCE TO _DINT
GET
nHeight REF= _nHeight;
END_GET
END_PROPERTY

PROPERTY PUBLIC nWidth : REFERENCE TO _DINT
GET
nWidth REF= _nWidth;
END_GET
END_PROPERTY

PROPERTY PUBLIC nX : REFERENCE TO _DINT
GET
nX REF= _nX;
END_GET
END_PROPERTY

PROPERTY PUBLIC nY : REFERENCE TO _DINT
GET
nY REF= _nY;
END_GET
END_PROPERTY

METHOD PROTECTED SetMemberReference
VAR_INPUT
END_VAR
_nX.MakeReferenceTo(activeData.nX);
_nY.MakeReferenceTo(activeData.nY);
_nWidth.MakeReferenceTo(activeData.nWidth);
_nHeight.MakeReferenceTo(activeData.nHeight);
END_METHOD

PROPERTY PUBLIC Size : UDINT
GET
Size := SIZEOF(activeData);
END_GET
END_PROPERTY

METHOD TryMakeReferenceTo : BOOL
VAR_INPUT
	Target : I_Datatype;
END_VAR
VAR
	pTargetData : POINTER TO TcVnRectangle_DINT;
END_VAR
IF NOT IsEquivalentTo(Target) THEN
	RETURN;
END_IF

pTargetData := Target.Address;
activeData REF= pTargetData^;
SetMemberReference();
TryMakeReferenceTo := TRUE;
END_METHOD

PROPERTY PUBLIC Value : REFERENCE TO TcVnRectangle_DINT
GET
Value REF= activeData;
END_GET
END_PROPERTY

END_FUNCTION_BLOCK

// ---- Datatypes/Structs/_TcVnRectangle_UDINT.TcPOU
{attribute 'linkalways'} 
{attribute 'no_explicit_call' := 'This FB is a CLASS and must be accessed using methods or properties'}
{attribute 'enable_dynamic_creation'}
FUNCTION_BLOCK _TcVnRectangle_UDINT EXTENDS StructuredDatatypeBase
VAR
	localData : TcVnRectangle_UDINT;
	activeData : REFERENCE TO TcVnRectangle_UDINT REF= localData;
	_nX : _UDINT(localData.nX);
	_nY : _UDINT(localData.nY);
    _nWidth : _UDINT(localData.nWidth);
	_nHeight : _UDINT(localData.nHeight);
END_VAR

PROPERTY PUBLIC Address : PVOID
GET
Address := ADR(activeData);
END_GET
END_PROPERTY

METHOD PUBLIC ClearReference
VAR_INPUT
END_VAR
activeData REF= localData;
SetMemberReference();
END_METHOD

METHOD PUBLIC Clone : I_Datatype
VAR
    pClone : POINTER TO _TcVnRectangle_UDINT;
END_VAR
pClone := __NEW(_TcVnRectangle_UDINT());
pClone^.Value := Value;
Clone := pClone^;
END_METHOD

METHOD FB_init : BOOL
VAR_INPUT
	bInitRetains : BOOL; // if TRUE, the retain variables are initialized (warm start / cold start)
	bInCopyCode : BOOL;  // if TRUE, the instance afterwards gets moved into the copy code (online change)
END_VAR
SetMemberReference();
AddMember('nX',_nX);
AddMember('nY',_nY);
AddMember('nWidth',_nWidth);
AddMember('nHeight',_nHeight);
END_METHOD

PROPERTY PUBLIC Identifier : T_MAXSTRING
GET
Identifier := 'TcVnRectangle_UDINT';
END_GET
END_PROPERTY

METHOD PUBLIC MakeReferenceTo
VAR_INPUT
	ReferenceTarget : REFERENCE TO TcVnRectangle_UDINT;
END_VAR
activeData REF= ReferenceTarget;
SetMemberReference();
END_METHOD

PROPERTY PUBLIC nHeight : REFERENCE TO _UDINT
GET
nHeight REF= _nHeight;
END_GET
END_PROPERTY

PROPERTY PUBLIC nWidth : REFERENCE TO _UDINT
GET
nWidth REF= _nWidth;
END_GET
END_PROPERTY

PROPERTY PUBLIC nX : REFERENCE TO _UDINT
GET
nX REF= _nX;
END_GET
END_PROPERTY

PROPERTY PUBLIC nY : REFERENCE TO _UDINT
GET
nY REF= _nY;
END_GET
END_PROPERTY

METHOD PROTECTED SetMemberReference
VAR_INPUT
END_VAR
_nX.MakeReferenceTo(activeData.nX);
_nY.MakeReferenceTo(activeData.nY);
_nWidth.MakeReferenceTo(activeData.nWidth);
_nHeight.MakeReferenceTo(activeData.nHeight);
END_METHOD

PROPERTY PUBLIC Size : UDINT
GET
Size := SIZEOF(activeData);
END_GET
END_PROPERTY

METHOD TryMakeReferenceTo : BOOL
VAR_INPUT
	Target : I_Datatype;
END_VAR
VAR
	pTargetData : POINTER TO TcVnRectangle_UDINT;
END_VAR
IF NOT IsEquivalentTo(Target) THEN
	RETURN;
END_IF

pTargetData := Target.Address;
activeData REF= pTargetData^;
SetMemberReference();
TryMakeReferenceTo := TRUE;
END_METHOD

PROPERTY PUBLIC Value : REFERENCE TO TcVnRectangle_UDINT
GET
Value REF= activeData;
END_GET
END_PROPERTY

END_FUNCTION_BLOCK

// ---- Datatypes/VisionDatatypePack.TcPOU
{attribute 'linkalways'} 
{attribute 'no_explicit_call' := 'This FB is a CLASS and must be accessed using methods or properties'}
{attribute 'enable_dynamic_creation'}
FUNCTION_BLOCK VisionDatatypePack
VAR
    // aliases
    _gVCP_REGISTER_ADDRESS : _GVCP_REGISTER_ADDRESS(0);
    _gVCP_REGISTER_VALUE : _GVCP_REGISTER_VALUE(0);
    _tcVnPoint : _TcVnPoint;
    _tcVnPoint2_DINT : _TcVnPoint2_DINT;
    _tcVnPoint2_LREAL : _TcVnPoint2_LREAL;
    _tcVnPoint2_REAL : _TcVnPoint2_REAL;
    _tcVnPoint3_LREAL : _TcVnPoint3_LREAL;
    _tcVnPoint3_REAL : _TcVnPoint3_REAL;
    _tcVnRectangle : _TcVnRectangle;
  
    _tcVnArray10_ITcVnImage : _TcVnArray10_ITcVnImage;
    _tcVnArray3_Point2_REAL : _TcVnArray3_Point2_REAL;
    _tcVnArray33_UDINT : _TcVnArray33_UDINT;
    _tcVnArray4_LREAL : _TcVnArray4_LREAL;
    _tcVnArray4_Point2_REAL : _TcVnArray4_Point2_REAL;
    _tcVnArray7_LREAL : _TcVnArray7_LREAL;
    _tcVnArray8_LREAL : _TcVnArray8_LREAL;
    _tcVnMatrix2x3_LREAL : _TcVnMatrix2x3_LREAL;
    _tcVnMatrix3x3_LREAL : _TcVnMatrix3x3_LREAL;
    _tcVnVector2_DINT : _TcVnVector2_DINT;
    _tcVnVector2_INT : _TcVnVector2_INT;
    _tcVnVector2_LREAL : _TcVnVector2_LREAL;
    _tcVnVector2_REAL : _TcVnVector2_REAL;
    _tcVnVector2_SINT : _TcVnVector2_SINT;
    _tcVnVector2_UINT : _TcVnVector2_UINT;
    _tcVnVector2_USINT : _TcVnVector2_USINT;
    _tcVnVector3_INT : _TcVnVector3_INT;
    _tcVnVector3_LREAL : _TcVnVector3_LREAL;
    _tcVnVector3_REAL : _TcVnVector3_REAL;
    _tcVnVector3_SINT : _TcVnVector3_SINT;
    _tcVnVector3_UINT : _TcVnVector3_UINT;
    _tcVnVector3_USINT : _TcVnVector3_USINT;
    _tcVnVector4_DINT : _TcVnVector4_DINT;
    _tcVnVector4_INT : _TcVnVector4_INT;
    _tcVnVector4_LREAL : _TcVnVector4_LREAL;
    _tcVnVector4_REAL : _TcVnVector4_REAL;
    _tcVnVector4_SINT : _TcVnVector4_SINT;
    _tcVnVector4_UINT : _TcVnVector4_UINT;
    _tcVnVector4_USINT : _TcVnVector4_USINT;
 
    // constants
    
    // arrays
    _array0to1OfDINT : _Array0to1OfDINT;
    _array0to1OfINT : _Array0to1OfINT;
    _array0to1OfLREAL : _Array0to1OfLREAL;
    _array0to1OfREAL : _Array0to1OfREAL;
    _array0to1OfSINT : _Array0to1OfSINT;
    _array0to1OfUINT : _Array0to1OfUINT;
    _array0to1OfUSINT : _Array0to1OfUSINT;
    _array0to2OfINT : _Array0to2OfINT;
    _array0to2OfLREAL : _Array0to2OfLREAL;
    _array0to2OfREAL : _Array0to2OfREAL;
    _array0to2OfSINT : _Array0to2OfSINT;
    _array0to2OfUINT : _Array0to2OfUINT;
    _array0to2OfUSINT : _Array0to2OfUSINT;
    _array0to3OfDINT : _Array0to3OfDINT;
    _array0to3OfINT : _Array0to3OfINT;
	_array0to3OfLREAL : _Array0to3OfLREAL;
    _array0to3OfREAL : _Array0to3OfREAL;
    _array0to6OfLREAL : _Array0to6OfLREAL;
    _array0to7OfLREAL : _Array0to7OfLREAL;
	_array0to1_0to2OfLREAL : _Array0to1_0to2OfLREAL;
	_array0to2_0to2OfLREAL : _Array0to2_0to2OfLREAL;
    
    // enums
	_eTcVn2dCodeSearchStrategy : _ETcVn2dCodeSearchStrategy(ETcVn2dCodeSearchStrategy.TCVN_CSS_DEFAULT);
    _eTcVnAdaptiveThresholdMethod : _ETcVnAdaptiveThresholdMethod(ETcVnAdaptiveThresholdMethod.TCVN_ATM_MEAN);
    _eTcVnBarcodeSearchDirection : _ETcVnBarcodeSearchDirection(ETcVnBarcodeSearchDirection.TCVN_BSD_ANY);
    _eTcVnBarcodeType : _ETcVnBarcodeType(ETcVnBarcodeType.TCVN_BT_CODABAR);
    _eTcVnBlobCombination : _ETcVnBlobCombination(ETcVnBlobCombination.TCVN_BC_SMALLEST);
    _eTcVnBoostClassifierType : _ETcVnBoostClassifierType(ETcVnBoostClassifierType.TCVN_BCT_DISCRETE);
    _eTcVnBorderInterpolationMethod : _ETcVnBorderInterpolationMethod(ETcVnBorderInterpolationMethod.TCVN_BIM_DEFAULT);
    _eTcVnCalibrationPattern : _ETcVnCalibrationPattern(ETcVnCalibrationPattern.TCVN_CP_CIRCLES_SYM);
    _eTcVnCalibrationPatternOrigin : _ETcVnCalibrationPatternOrigin(ETcVnCalibrationPatternOrigin.TCVN_CPO_TOPCENTER);
    _eTcVnCameraState : _ETcVnCameraState(ETcVnCameraState.TCVN_CS_INITIAL);
    _eTcVnClusteringAlgorithm : _ETcVnClusteringAlgorithm(ETcVnClusteringAlgorithm.TCVN_CA_KMEANSPP);
	_eTcVnCodeDetectionModel : _ETcVnCodeDetectionModel(ETcVnCodeDetectionModel.TCVN_CDM_DETECT_1_1);
	_eTcVnCodeType : _ETcVnCodeType(ETcVnCodeType.TCVN_CT_ANY);
    _eTcVnColorMap : _ETcVnColorMap(ETcVnColorMap.TCVN_CM_AUTUMN);
    _eTcVnColorMapSize : _ETcVnColorMapSize(ETcVnColorMapSize.TCVN_CMS_256);
    _eTcVnColorSpaceTransform : _ETcVnColorSpaceTransform(ETcVnColorSpaceTransform.TCVN_CST_RGBA_TO_RGB);
    _eTcVnColorTrainingMethod : _ETcVnColorTrainingMethod(ETcVnColorTrainingMethod.TCVN_CTM_LAB);
    _eTcVnConnectedComponentsAlgorithm : _ETcVnConnectedComponentsAlgorithm(ETcVnConnectedComponentsAlgorithm.TCVN_CCA_WU);
    _eTcVnContainerExportFormat : _ETcVnContainerExportFormat(ETcVnContainerExportFormat.TCVN_CEF_XML);
    _eTcVnContourApproximationMethod : _ETcVnContourApproximationMethod(ETcVnContourApproximationMethod.TCVN_CAM_NONE);
    _eTcVnContourRetrievalMode : _ETcVnContourRetrievalMode(ETcVnContourRetrievalMode.TCVN_CRM_EXTERNAL);
    _eTcVnContoursMatchComparisonMethod : _ETcVnContoursMatchComparisonMethod(ETcVnContoursMatchComparisonMethod.TCVN_CMCM_CONTOURS_MATCH_I1);
    _eTcVnDiffusivityTypeKAZE : _ETcVnDiffusivityTypeKAZE(ETcVnDiffusivityTypeKAZE.TCVN_DT1_KAZE_PM_G1);
    _eTcVnDistanceTransformationLabel : _ETcVnDistanceTransformationLabel(ETcVnDistanceTransformationLabel.TCVN_DTL_CCOMP);
    _eTcVnDistanceTransformationMask : _ETcVnDistanceTransformationMask(ETcVnDistanceTransformationMask.TCVN_DTM_PRECISE);
    _eTcVnDistanceType : _ETcVnDistanceType(ETcVnDistanceType.TCVN_DT_USER);
    _eTcVnDrawMatchesFlags : _ETcVnDrawMatchesFlags(ETcVnDrawMatchesFlags.TCVN_DMF_DEFAULT);
    _eTcVnDrawShape : _ETcVnDrawShape(ETcVnDrawShape.TCVN_DS_CIRCLE);
    _eTcVnEdgeDetectionAlgorithm : _ETcVnEdgeDetectionAlgorithm(ETcVnEdgeDetectionAlgorithm.TCVN_EDA_INTERPOLATION);
    _eTcVnEdgeDirection : _ETcVnEdgeDirection(ETcVnEdgeDirection.TCVN_ED_DARK_TO_LIGHT);
    _eTcVnElementType : _ETcVnElementType(ETcVnElementType.TCVN_ET_SAME_AS_SOURCE);
    _eTcVnEstimationAlgorithm : _ETcVnEstimationAlgorithm(ETcVnEstimationAlgorithm.TCVN_EA_DEFAULT);
    _eTcVnExtremePointDirection : _ETcVnExtremePointDirection(ETcVnExtremePointDirection.TCVN_EPD_TOP_LEFT);
    _eTcVnFeatureDescriptorTypeAKAZE : _ETcVnFeatureDescriptorTypeAKAZE(ETcVnFeatureDescriptorTypeAKAZE.TCVN_FDT_AKAZE_KAZE_UPRIGHT);
    _eTcVnFeatureScalingType : _ETcVnFeatureScalingType(ETcVnFeatureScalingType.TCVN_FST1_MAXABS);
    _eTcVnFeatureScoreTypeORB : _ETcVnFeatureScoreTypeORB(ETcVnFeatureScoreTypeORB.TCVN_FST_ORB_HARRIS);
    _eTcVnFilterDirection : _ETcVnFilterDirection(ETcVnFilterDirection.TCVN_FD_X);
	_eTcVnFindTemplateWalshOptions : _ETcVnFindTemplateWalshOptions(ETcVnFindTemplateWalshOptions.TCVN_FTWO_NONE);
    _eTcVnFlipAxis : _ETcVnFlipAxis(ETcVnFlipAxis.TCVN_FA_X);
    _eTcVnFontType : _ETcVnFontType(ETcVnFontType.TCVN_FT_HERSHEY_SIMPLEX);
    _eTcVnHoughMethod : _ETcVnHoughMethod(ETcVnHoughMethod.TCVN_HM_STANDARD);
    _eTcVnInitializableFunction : _ETcVnInitializableFunction(ETcVnInitializableFunction.TCVN_IF_OCR);
    _eTcVnInterpolationType : _ETcVnInterpolationType(ETcVnInterpolationType.TCVN_IT_NEAREST_NEIGHBOR);
    _eTcVnKeypointDetectionTypeAGAST : _ETcVnKeypointDetectionTypeAGAST(ETcVnKeypointDetectionTypeAGAST.TCVN_KDT_AGAST_5_8);
    _eTcVnKeypointDetectionTypeFAST : _ETcVnKeypointDetectionTypeFAST(ETcVnKeypointDetectionTypeFAST.TCVN_KDT_FAST_5_8);
    _eTcVnKnn : _ETcVnKnn(ETcVnKnn.TCVN_KNN_CLASSIFIER);
    _eTcVnLineType : _ETcVnLineType(ETcVnLineType.TCVN_LT_4_CONNECTED);
	_eTcVnMatchTemplateWalshOptions : _ETcVnMatchTemplateWalshOptions(ETcVnMatchTemplateWalshOptions.TCVN_MTWO_NONE);
    _eTcVnMorphologicalOperator : _ETcVnMorphologicalOperator(ETcVnMorphologicalOperator.TCVN_MO_EROSION);
    _eTcVnNbc : _ETcVnNbc(ETcVnNbc.TCVN_NBC_CLASSIFIER);
    _eTcVnNormalizationType : _ETcVnNormalizationType(ETcVnNormalizationType.TCVN_NT_INF);
    _eTcVnOcrModelType : _ETcVnOcrModelType(ETcVnOcrModelType.TCVN_OMT_NUMBERS);
    _eTcVnOcrOptions : _ETcVnOcrOptions(ETcVnOcrOptions.TCVN_OO_NONE);
    _eTcVnOrientationMethod : _ETcVnOrientationMethod(ETcVnOrientationMethod.TCVN_OM_PCA);
    _eTcVnPaddingMode : _ETcVnPaddingMode(ETcVnPaddingMode.TCVN_PM_NONE);
    _eTcVnPixelConnectivity : _ETcVnPixelConnectivity(ETcVnPixelConnectivity.TCVN_PC_4);
    _eTcVnPixelEncoding : _ETcVnPixelEncoding(ETcVnPixelEncoding.TCVN_PE_NONE);
    _eTcVnPixelPackMode : _ETcVnPixelPackMode(ETcVnPixelPackMode.TCVN_PPM_NONE);
    _eTcVnPrototypeClusterer : _ETcVnPrototypeClusterer(ETcVnPrototypeClusterer.TCVN_PC_NOVELTY_DETECTOR);
    _eTcVnRectangleIntersection : _ETcVnRectangleIntersection(ETcVnRectangleIntersection.TCVN_RI_NONE);
    _eTcVnRotationAngle : _ETcVnRotationAngle(ETcVnRotationAngle.TCVN_RA_90_DEG);
    _eTcVnRTrees : _ETcVnRTrees(ETcVnRTrees.TCVN_RT_CLASSIFIER);
    _eTcVnSignedNormalization : _ETcVnSignedNormalization(ETcVnSignedNormalization.TCVN_SN_FIX_ZERO);
    _eTcVnSolvePnPMethod : _ETcVnSolvePnPMethod(ETcVnSolvePnPMethod.TCVN_SPM_ITERATIVE);
    _eTcVnSta : _ETcVnSta(ETcVnSta.TCVN_STA_CLASSIFIER);
    _eTcVnStructuringElementShape : _ETcVnStructuringElementShape(ETcVnStructuringElementShape.TCVN_SES_RECTANGLE);
    _eTcVnSvm : _ETcVnSvm(ETcVnSvm.TCVN_SVM_C_CLASSIFIER);
    _eTcVnSvmKernelType : _ETcVnSvmKernelType(ETcVnSvmKernelType.TCVN_SKT_LINEAR);
    _eTcVnSvmSgdClassifierMarginType : _ETcVnSvmSgdClassifierMarginType(ETcVnSvmSgdClassifierMarginType.TCVN_SSCMT_SOFT_MARGIN);
    _eTcVnSvmSgdClassifierType : _ETcVnSvmSgdClassifierType(ETcVnSvmSgdClassifierType.TCVN_SSCT_SGD);
    _eTcVnTemplateMatchMethod : _ETcVnTemplateMatchMethod(ETcVnTemplateMatchMethod.TCVN_TMM_SQDIFF);
    _eTcVnThresholdType : _ETcVnThresholdType(ETcVnThresholdType.TCVN_TT_BINARY);
    _eTcVnTimestamp : _ETcVnTimestamp(ETcVnTimestamp.TCVN_TS_IMAGE_COMPLETED);
    _eTcVnVectorCompareMethod : _ETcVnVectorCompareMethod(ETcVnVectorCompareMethod.TCVN_VCM_EUCLIDEAN);
    _eTcVnWorldCoordinateSystem : _ETcVnWorldCoordinateSystem(ETcVnWorldCoordinateSystem.TCVN_WCS_X_RIGHT_Y_DOWN);
    _eTcWatchdogAccumulationType : _ETcWatchdogAccumulationType(ETcWatchdogAccumulationType.WD_ACC_TYPE_MEAN);
    _gEV_CAMERA_STATE : _GEV_CAMERA_STATE(GEV_CAMERA_STATE.GEV_CAMERA_IDLE);
    _eTcVnDataLayout : _ETcVnDataLayout(ETcVnDataLayout.TCVN_DL_DEFAULT);
    _eTcVnReduceType : _ETcVnReduceType(ETcVnReduceType.TCVN_RT_REDUCE_SUM);
    _eTcVnCircularityCalculationMethod : _ETcVnCircularityCalculationMethod(ETcVnCircularityCalculationMethod.TCVN_CCM_DEFAULT);
    _eTcVnDataMatrixOptions : _ETcVnDataMatrixOptions(ETcVnDataMatrixOptions.TCVN_DMO_DEFAULT);
    _eTcVnLayerNameType : _ETcVnLayerNameType(ETcVnLayerNameType.TCVN_LNT_ALL);
	
    _eTcVnComparisonOperator : _ETcVnComparisonOperator(ETcVnComparisonOperator.TCVN_CO_LESS);
    _eTcVnDetectBarcodesWalshOptions : _ETcVnDetectBarcodesWalshOptions(ETcVnDetectBarcodesWalshOptions.TCVN_DBWO_HORIZONTAL);
    _eTcVnDetectPatternPointsOptions : _ETcVnDetectPatternPointsOptions(ETcVnDetectPatternPointsOptions.TCVN_DPPO_SYMMETRIC);
    _eTcVnDotCodeOptions : _ETcVnDotCodeOptions(ETcVnDotCodeOptions.TCVN_DCO_DEFAULT);
    _eTcVnEdgeSelection : _ETcVnEdgeSelection(ETcVnEdgeSelection.TCVN_ES_RISING);
    _eTcVnFindRoisMethod : _ETcVnFindRoisMethod(ETcVnFindRoisMethod.TCVN_FRM_GRID);
    _eTcVnJpegSampling : _ETcVnJpegSampling(ETcVnJpegSampling.TCVN_JS_444);
    _eTcVnMergeRegionsOptions : _ETcVnMergeRegionsOptions(ETcVnMergeRegionsOptions.TCVN_MRO_UPRIGHT_BOUNDING_RECT);
    _eTcVnPolarizedImageInterpolation : _ETcVnPolarizedImageInterpolation(ETcVnPolarizedImageInterpolation.TCVN_PII_NONE);
    _eTcVnSalientFeaturesMethod : _ETcVnSalientFeaturesMethod(ETcVnSalientFeaturesMethod.TCVN_SFM_WALSH_CODE);
    // structs
    _gVSP_IMAGE_INFO : _GVSP_IMAGE_INFO;
    _gVSP_LEADER_PAYLOAD_IMAGE : _GVSP_LEADER_PAYLOAD_IMAGE;
    _gVSP_PIXEL_FORMAT : _GVSP_PIXEL_FORMAT;
    _tcVnCameraCalibrationOptions : _TcVnCameraCalibrationOptions;
    _tcVnCircularArc : _TcVnCircularArc;
    _tcVnCodeGrades1D : _TcVnCodeGrades1D;
    _tcVnCodeGradesDM : _TcVnCodeGradesDM;
    _tcVnCodeGradesQR : _TcVnCodeGradesQR;
    _tcVnDMatch : _TcVnDMatch;
	_tcVnImageInfo : _TcVnImageInfo;
    _tcVnKeyPoint : _TcVnKeyPoint;
//  _tcVnMatrix : _TcVnMatrix;
    _tcVnMoments : _TcVnMoments;
    _tcVnParamsAGAST : _TcVnParamsAGAST;
    _tcVnParamsAKAZE : _TcVnParamsAKAZE;
    _tcVnParamsBlobDetection : _TcVnParamsBlobDetection;
    _tcVnParamsBRISK : _TcVnParamsBRISK;
    _tcVnParamsFAST : _TcVnParamsFAST;
    _tcVnParamsGFTT : _TcVnParamsGFTT;
    _tcVnParamsKAZE : _TcVnParamsKAZE;
    _tcVnParamsMSER : _TcVnParamsMSER;
    _tcVnParamsORB : _TcVnParamsORB;
    _tcVnParamsSB : _TcVnParamsSB;
    _tcVnPixelFormat : _TcVnPixelFormat;
	_tcVnRectangle_DINT : _TcVnRectangle_DINT;
    _tcVnRectangle_UDINT : _TcVnRectangle_UDINT;
    _tcVnRotatedRectangle : _TcVnRotatedRectangle;
    _tcVnSize2_REAL : _TcVnSize2_REAL;
	
    _gVCP_ADDRESS_VALUE_PAIR : _GVCP_ADDRESS_VALUE_PAIR;
    _tcVnSize2_DINT : _TcVnSize2_DINT;
    _tcVnParamsFindRois : _TcVnParamsFindRois;
    _tcVnParamsWalshBarcodeDetection : _TcVnParamsWalshBarcodeDetection;
	// interfaces
	_iTcVnImage : _ITcVnImage;
	_iTcVnContainer : _ITcVnContainer;
	_iTcVnDisplayableImage : _ITcVnDisplayableImage;
	
END_VAR

METHOD RegisterWithDatatypes
VAR_INPUT
	Datatypes : I_Datatypes;
END_VAR
// aliases
Datatypes.RegisterDatatype(_GVCP_REGISTER_ADDRESS);
Datatypes.RegisterDatatype(_gVCP_REGISTER_VALUE);
Datatypes.RegisterDatatype(_tcVnPoint);
Datatypes.RegisterDatatype(_tcVnPoint2_DINT);
Datatypes.RegisterDatatype(_tcVnPoint2_LREAL);
Datatypes.RegisterDatatype(_tcVnPoint2_REAL);
Datatypes.RegisterDatatype(_tcVnPoint3_LREAL);
Datatypes.RegisterDatatype(_tcVnPoint3_REAL);
Datatypes.RegisterDatatype(_tcVnRectangle);

Datatypes.RegisterDatatype(_tcVnArray10_ITcVnImage);
Datatypes.RegisterDatatype(_tcVnArray3_Point2_REAL);
Datatypes.RegisterDatatype(_tcVnArray33_UDINT);
Datatypes.RegisterDatatype(_tcVnArray4_LREAL);
Datatypes.RegisterDatatype(_tcVnArray4_Point2_REAL);
Datatypes.RegisterDatatype(_tcVnArray7_LREAL);
Datatypes.RegisterDatatype(_tcVnArray8_LREAL);
Datatypes.RegisterDatatype(_tcVnMatrix2x3_LREAL);
Datatypes.RegisterDatatype(_tcVnMatrix3x3_LREAL);
Datatypes.RegisterDatatype(_tcVnVector2_DINT);
Datatypes.RegisterDatatype(_tcVnVector2_INT);
Datatypes.RegisterDatatype(_tcVnVector2_LREAL);
Datatypes.RegisterDatatype(_tcVnVector2_REAL);
Datatypes.RegisterDatatype(_tcVnVector2_SINT);
Datatypes.RegisterDatatype(_tcVnVector2_UINT);
Datatypes.RegisterDatatype(_tcVnVector2_USINT);
Datatypes.RegisterDatatype(_tcVnVector3_INT);
Datatypes.RegisterDatatype(_tcVnVector3_LREAL);
Datatypes.RegisterDatatype(_tcVnVector3_REAL);
Datatypes.RegisterDatatype(_tcVnVector3_SINT);
Datatypes.RegisterDatatype(_tcVnVector3_UINT);
Datatypes.RegisterDatatype(_tcVnVector3_USINT);
Datatypes.RegisterDatatype(_tcVnVector4_DINT);
Datatypes.RegisterDatatype(_tcVnVector4_INT);
Datatypes.RegisterDatatype(_tcVnVector4_LREAL);
Datatypes.RegisterDatatype(_tcVnVector4_REAL);
Datatypes.RegisterDatatype(_tcVnVector4_SINT);
Datatypes.RegisterDatatype(_tcVnVector4_UINT);
Datatypes.RegisterDatatype(_tcVnVector4_USINT);

// constants

// arrays
Datatypes.RegisterDatatype(_array0to1OfDINT);
Datatypes.RegisterDatatype(_array0to1OfINT);
Datatypes.RegisterDatatype(_array0to1OfLREAL);
Datatypes.RegisterDatatype(_array0to1OfREAL);
Datatypes.RegisterDatatype(_array0to1OfSINT);
Datatypes.RegisterDatatype(_array0to1OfUINT);
Datatypes.RegisterDatatype(_array0to1OfUSINT);
Datatypes.RegisterDatatype(_array0to2OfINT);
Datatypes.RegisterDatatype(_array0to2OfLREAL);
Datatypes.RegisterDatatype(_array0to2OfREAL);
Datatypes.RegisterDatatype(_array0to2OfSINT);
Datatypes.RegisterDatatype(_array0to2OfUINT);
Datatypes.RegisterDatatype(_array0to2OfUSINT);
Datatypes.RegisterDatatype(_array0to3OfDINT);
Datatypes.RegisterDatatype(_array0to3OfINT);
Datatypes.RegisterDatatype(_array0to3OfLREAL);
Datatypes.RegisterDatatype(_array0to3OfREAL);
Datatypes.RegisterDatatype(_array0to6OfLREAL);
Datatypes.RegisterDatatype(_array0to7OfLREAL);
Datatypes.RegisterDatatype(_array0to1_0to2OfLREAL);
Datatypes.RegisterDatatype(_array0to2_0to2OfLREAL);

